(* CODESYS project CtaAppStellAntrieb_1.0.0.3.library
   Description: Stell- Antriebs Library der CTA
   Version: 1.0.0.3
   Title: CtaAppStellAntrieb
   Author: SIS
   Company: CTA
   DocFormat: reStructuredText
   Placeholder: CtaAppStellAntrieb
   DefaultNamespace: CtaAppStellAntrieb
   CompiledLibraryCompatibilityVersion: CODESYS V3.5 SP16 Patch 3
   LanguageModelAttribute: qualified-access-only

Project tree, tasks and I/O mapping:
  libraries: Standard, 3.5.18.0 (System); CtaAppBasic, 1.0.0.0 (CTA); CtaAppBmk, 1.0.0.0 (CTA); CtaAppReport, 1.0.0.0 (CTA); CtaSysConfig, 1.0.0.2 (CTA); VisuDialogs, 3.5.16.20 (System); VisuSymbols, 4.5.0.0 (System); CtaSysMotor, 1.0.0.0 (CTA); CtaVisSymbols, 1.0.0.0 (CTA); CtaAppDumper, 1.0.0.0 (CTA); CtaSysIO, 1.0.0.1 (CTA); CtaAppInfluxLog, 1.0.0.1 (CTA); CtaAppModbusSpezifikation, 1.0.0.0 (CTA); CtaVisHelp, 1.0.0.0 (CTA)
  40 Visualizations/
    COLLECTOR/
      visualisation StellAntrieb_Collector
      visualisation StellAntrieb_Collector_TEMP
      Help Funktionen/
        visualisation SelSort
        visualisation SortPfeil
    ICON/
      StellAntrieb_RIGHT/
        Motor_Right/
          Valve_Mix/
            Above/
              visualisation StellAntrieb_MR_Valve_Mix_RA_CheckEnabled
              visualisation StellAntrieb_MR_Valve_Mix_RA_CheckQuerry
              visualisation StellAntrieb_MR_Valve_Mix_Txt_R_Above
            Below/
              visualisation StellAntrieb_MR_Valve_Mix_RB_CheckEnabled
              visualisation StellAntrieb_MR_Valve_Mix_RB_CheckQuerry
              visualisation StellAntrieb_MR_Valve_Mix_Txt_R_Below
          Valve_Flow/
            Above/
              visualisation StellAntrieb_MR_Valve_Flow_RA_CheckEnabled
              visualisation StellAntrieb_MR_Valve_Flow_RA_CheckQuerry
              visualisation StellAntrieb_MR_Valve_Flow_Txt_R_Above
            Below/
              visualisation StellAntrieb_MR_Valve_Flow_RB_CheckEnabled
              visualisation StellAntrieb_MR_Valve_Flow_RB_CheckQuerry
              visualisation StellAntrieb_MR_Valve_Flow_Txt_R_Below
          Valve_AB_Down/
            Above/
              visualisation StellAntrieb_MR_Valve_AB_Down_RA_CheckQuerry
              visualisation StellAntrieb_MR_Valve_AB_Down_Txt_R_Above
              visualisation StellAntrieb_MR_Valve_AB_Down_RA_CheckEnabled
            Below/
              visualisation StellAntrieb_MR_Valve_AB_Down_Txt_R_Below
              visualisation StellAntrieb_MR_Valve_AB_Down_RB_CheckEnabled
              visualisation StellAntrieb_MR_Valve_AB_Down_RB_CheckQuerry
          Valve_AB_Up/
            Above/
              visualisation StellAntrieb_MR_Valve_AB_Up_RA_CheckEnabled
              visualisation StellAntrieb_MR_Valve_AB_Up_RA_CheckQuerry
              visualisation StellAntrieb_MR_Valve_AB_Up_Txt_R_Above
            Below/
              visualisation StellAntrieb_MR_Valve_AB_Up_RB_CheckEnabled
              visualisation StellAntrieb_MR_Valve_AB_Up_RB_CheckQuerry
              visualisation StellAntrieb_MR_Valve_AB_Up_Txt_R_Below
        Motor_Above/
          Valve_AB_Left/
            visualisation StellAntrieb_MA_Valve_AB_Left_RA_CheckEnabled
            visualisation StellAntrieb_MA_Valve_AB_Left_RA_CheckQuerry
            visualisation StellAntrieb_MA_Valve_AB_Left_Txt_R_Above
          Valve_AB_Right/
            visualisation StellAntrieb_MA_Valve_AB_Right_RA_CheckEnabled
            visualisation StellAntrieb_MA_Valve_AB_Right_RA_CheckQuerry
            visualisation StellAntrieb_MA_Valve_AB_Right_Txt_R_Above
          Valve_Flow/
            visualisation StellAntrieb_MA_Valve_Flow_RA_CheckEnabled
            visualisation StellAntrieb_MA_Valve_Flow_RA_CheckQuerry
            visualisation StellAntrieb_MA_Valve_Flow_Txt_R_Above
          Valve_Mix/
            visualisation StellAntrieb_MA_Valve_Mix_RA_CheckEnabled
            visualisation StellAntrieb_MA_Valve_Mix_RA_CheckQuerry
            visualisation StellAntrieb_MA_Valve_Mix_Txt_R_Above
        Motor_Below/
          Valve_AB_Right/
            visualisation StellAntrieb_MB_Valve_AB_Right_RB_CheckEnabled
            visualisation StellAntrieb_MB_Valve_AB_Right_RB_CheckQuerry
            visualisation StellAntrieb_MB_Valve_AB_Right_Txt_R_Below
          Valve_AB_Left/
            visualisation StellAntrieb_MB_Valve_AB_Left_RB_CheckEnabled
            visualisation StellAntrieb_MB_Valve_AB_Left_RB_CheckQuerry
            visualisation StellAntrieb_MB_Valve_AB_Left_Txt_R_Below
          Valve_Flow/
            visualisation StellAntrieb_MB_Valve_Flow_RB_CheckEnabled
            visualisation StellAntrieb_MB_Valve_Flow_RB_CheckQuerry
            visualisation StellAntrieb_MB_Valve_Flow_Txt_R_Below
          Valve_Mix/
            visualisation StellAntrieb_MB_Valve_Mix_RB_CheckEnabled
            visualisation StellAntrieb_MB_Valve_Mix_RB_CheckQuerry
            visualisation StellAntrieb_MB_Valve_Mix_Txt_R_Below
      StellAntrieb_BASE/
        Ventile/
          DurchflussVentil/
            Motor_Below/
              visualisation MB_Durchgang
            Motor_Above/
              visualisation MA_Durchgang
            Motor_Right/
              visualisation MR_Durchgang
            Motor_Left/
              visualisation ML_Durchgang
          DreiWegVentil/
            Motor_Below/
              visualisation MB_Ventil_AB_L
              visualisation MB_Ventil_Verteiler
              visualisation MB_Ventil_AB_R
            Motor_Above/
              visualisation MA_Ventil_AB_L
              visualisation MA_Ventil_Verteiler
              visualisation MA_Ventil_AB_R
            Motor_Right/
              visualisation MR_Ventil_AB_Up
              visualisation MR_Ventil_Verteiler
              visualisation MR_Ventil_AB_Down
            Motor_Left/
              visualisation ML_Ventil_AB_Down
              visualisation ML_Ventil_Verteiler
              visualisation ML_Ventil_AB_Up
        Icons/
          visualisation Motor
          Motor_Left/
            visualisation Icon_ML_AB_Down
            visualisation Icon_ML_AB_Up
            visualisation Icon_ML_Verteiler
            visualisation Icon_ML_Durchfluss
          Motor_Right/
            visualisation Icon_MR_AB_Down
            visualisation Icon_MR_AB_Up
            visualisation Icon_MR_Durchfluss
            visualisation Icon_MR_Verteiler
          Motor_Below/
            visualisation Icon_MB_AB_L
            visualisation Icon_MB_AB_R
            visualisation Icon_MB_Verteiler
            visualisation Icon_MB_Durchfluss
          Motor_Above/
            visualisation Icon_MA_AB_L
            visualisation Icon_MA_AB_R
            visualisation Icon_MA_Durchfluss
            visualisation Icon_MA_Verteiler
        Value/
          visualisation ValueUpDwn
          visualisation ValueDwnUp
      StellAntrieb_LEFT/
        Motor_LEFT/
          Valve_AB_Down/
            Above/
              visualisation StellAntrieb_ML_Valve_AB_Down_LA_CheckEnabled
              visualisation StellAntrieb_ML_Valve_AB_Down_LA_CheckQuerry
              visualisation StellAntrieb_ML_Valve_AB_Down_Txt_L_Above
            Below/
              visualisation StellAntrieb_ML_Valve_AB_Down_LB_CheckEnabled
              visualisation StellAntrieb_ML_Valve_AB_Down_LB_CheckQuerry
              visualisation StellAntrieb_ML_Valve_AB_Down_Txt_L_Below
          Valve_Mix/
            Above/
              visualisation StellAntrieb_ML_Valve_Mix_LA_CheckEnabled
              visualisation StellAntrieb_ML_Valve_Mix_LA_CheckQuerry
              visualisation StellAntrieb_ML_Valve_Mix_Txt_L_Above
            Below/
              visualisation StellAntrieb_ML_Valve_Mix_LB_CheckEnabled
              visualisation StellAntrieb_ML_Valve_Mix_LB_CheckQuerry
              visualisation StellAntrieb_ML_Valve_Mix_Txt_L_Below
          Valve_Flow/
            Above/
              visualisation StellAntrieb_ML_Valve_Flow_LA_CheckEnabled
              visualisation StellAntrieb_ML_Valve_Flow_LA_CheckQuerry
              visualisation StellAntrieb_ML_Valve_Flow_Txt_L_Above
            Below/
              visualisation StellAntrieb_ML_Valve_Flow_LB_CheckEnabled
              visualisation StellAntrieb_ML_Valve_Flow_LB_CheckQuerry
              visualisation StellAntrieb_ML_Valve_Flow_Txt_L_Below
          Valve_AB_Up/
            Above/
              visualisation StellAntrieb_ML_Valve_AB_Up_LA_CheckEnabled
              visualisation StellAntrieb_ML_Valve_AB_Up_LA_CheckQuerry
              visualisation StellAntrieb_ML_Valve_AB_Up_Txt_L_Above
            Below/
              visualisation StellAntrieb_ML_Valve_AB_Up_LB_CheckEnabled
              visualisation StellAntrieb_ML_Valve_AB_Up_LB_CheckQuerry
              visualisation StellAntrieb_ML_Valve_AB_Up_Txt_L_Below
        Motor_Above/
          Valve_AB_Left/
            visualisation StellAntrieb_MA_Valve_AB_Left_LA_CheckEnabled
            visualisation StellAntrieb_MA_Valve_AB_Left_LA_CheckQuerry
            visualisation StellAntrieb_MA_Valve_AB_Left_Txt_L_Above
          Valve_AB_Right/
            visualisation StellAntrieb_MA_Valve_AB_Right_LA_CheckEnabled
            visualisation StellAntrieb_MA_Valve_AB_Right_Txt_L_Above
            visualisation StellAntrieb_MA_Valve_AB_Right_LA_CheckQuerry
          Valve_Flow/
            visualisation StellAntrieb_MA_Valve_Flow_Txt_L_Above
            visualisation StellAntrieb_MA_Valve_Flow_LA_CheckQuerry
            visualisation StellAntrieb_MA_Valve_Flow_LA_CheckEnabled
          Valve_Mix/
            visualisation StellAntrieb_MA_Valve_Mix_LA_CheckEnabled
            visualisation StellAntrieb_MA_Valve_Mix_LA_CheckQuerry
            visualisation StellAntrieb_MA_Valve_Mix_Txt_L_Above
        Motor_Below/
          Valve_AB_Left/
            visualisation StellAntrieb_MB_Valve_AB_Left_LB_CheckEnabled
            visualisation StellAntrieb_MB_Valve_AB_Left_LB_CheckQuerry
            visualisation StellAntrieb_MB_Valve_AB_Left_Txt_L_Below
          Valve_AB_Right/
            visualisation StellAntrieb_MB_Valve_AB_Right_LB_CheckEnabled
            visualisation StellAntrieb_MB_Valve_AB_Right_LB_CheckQuerry
            visualisation StellAntrieb_MB_Valve_AB_Right_Txt_L_Below
          Valve_Flow/
            visualisation StellAntrieb_MB_Valve_Flow_LB_CheckEnabled
            visualisation StellAntrieb_MB_Valve_Flow_LB_CheckQuerry
            visualisation StellAntrieb_MB_Valve_Flow_Txt_L_Below
          Valve_Mix/
            visualisation StellAntrieb_MB_Valve_Mix_LB_CheckEnabled
            visualisation StellAntrieb_MB_Valve_Mix_LB_CheckQuerry
            visualisation StellAntrieb_MB_Valve_Mix_Txt_L_Below
    POPUP/
      visualisation StellAntrieb_POPUP
      PARAMETER/
        visualisation StellAntrieb_PARAMETER
        visualisation StellAntrieb_ParameterListe
        StellAntrieb_ParameterBase/
          visualisation StellAntrieb_ParameterBase0
          visualisation StellAntrieb_ParameterBase
          visualisation StellAntrieb_ParameterBase2
          visualisation StellAntrieb_ParameterBase1
        StellAntrieb_Fuse/
          visualisation StellAntrieb_ParameterFuses0
          visualisation StellAntrieb_ParameterFuses
        StellAntrieb_IO/
          visualisation StellAntrieb_ParameterIO0
          visualisation StellAntrieb_ParameterIO1
          visualisation StellAntrieb_ParameterIO
          visualisation StellAntrieb_ParameterIO2
          visualisation StellAntrieb_ParameterIO3
          visualisation StellAntrieb_ParameterIO4
        StellAntrieb_InfluxDb/
          visualisation StellAntrieb_ParameterInfluxDb
          visualisation StellAntrieb_ParameterInfluxDb0
        visualisation StellAntrieb_Icon_StellAntrieb
        visualisation StellAntrieb_POPUP_IO_ITF
      visualisation StellAntrieb_PopUpListe
      MANUAL/
        visualisation StellAntrieb_MANUAL
      OVERVIEW/
        visualisation StellAntrieb_OVERVIEW
      BUS/
        visualisation StellAntrieb_BUS
        visualisation StellAntrieb_BUS_SW0_Detail
        visualisation StellAntrieb_BUS_CW0_Detail
        visualisation StellAntrieb_BUS_CS
        visualisation StellAntrieb_BUS_SW1_Detail
        visualisation StellAntrieb_BUS_SW2_Detail
      REPORTS/
        visualisation StellAntrieb_REPORTS
      IO/
        visualisation StellAntrieb_IO0
        visualisation StellAntrieb_IO
        visualisation StellAntrieb_IO1
  30 Program Organization Units/
    function block fbStellAantrieb [ST]: proHandOn, proAuto, proHandOff, proHandOnY, proHardWareHandModulAktive, actConfig, p_scInfluxDb_fbxEnable, p_scActuatorFuse_fbxEnable, p_scActuatorFuse_fbxInputMb, p_scActuatorFuse_fbxDoesAlarm, p_scBase_fbxEnable, p_scBase_fbxControllMb, p_scBase_fbxInvertiert, p_scBase_fbxRegulatet, p_scBase_fbrYMin, p_scBase_fbrYMax, p_scBase_fbxEnStartPosition, p_scBase_fbrYStartPos, p_scBase_fbtStartPosTime, p_scBase_fbrYStopp, p_scBase_fbtYSettingTime, p_scBase_fbxEnDigitalValve, p_scBase_fbrHysteresisDigital, p_scBase_fbrRefIsOpen, p_scBase_fbrRefIsClosed, p_scBase_fbxEnDigitalMonitoring, p_scBase_fbxEnAnalogMonitoring, p_scFuse_fbxEnable, p_scFuse_fbxInputMb, p_scFuse_fbxDoesAlarm, p_scInStellAtRevisionSwitch_fbxEnable, p_scInStellAtRevisionSwitch_fbxInputMb, p_scInStellAtReady_fbxEnable, p_scInStellAtReady_fbxInputMb, p_scInStellAtHand_fbxEnable, p_scInStellAtHand_fbxInputMb, p_scInStellAtRükClosed_fbxEnable, p_scInStellAtRükClosed_fbxInputMb, p_scInStellAtRükClosed_fbxDoesAlarm, p_scInStellAtRükClosed_fbtDelayStart, p_scInStellAtRükClosed_fbtDelayRun, p_scInStellAtRükClosed_fbiTypeOfAck, p_scInStellAtRükClosed_fbiMaxErrorRetryAllowed, p_scInStellAtRükOpen_fbxEnable, p_scInStellAtRükOpen_fbxInputMb, p_scInStellAtRükOpen_fbxDoesAlarm, p_scInStellAtRükOpen_fbtDelayStart, p_scInStellAtRükOpen_fbtDelayRun, p_scInStellAtRükOpen_fbiTypeOfAck, p_scInStellAtRükOpen_fbiMaxErrorRetryAllowed, p_scInStellAtActualPosition_fbxEnable, p_scInStellAtActualPosition_fbxInputMb, p_scInStellAtActualPosition_fbxDoesAlarm, p_scInStellAtActualPosition_fbrMaxDiff, p_scInStellAtActualPosition_fbtDelayStart, p_scInStellAtActualPosition_fbtDelayRun, p_scInStellAtActualPosition_fbiTypeOfAck, p_scInStellAtActualPosition_fbiMaxErrorRetryAllowed, p_scManual_fbxAlowManualOn, p_scManual_fbuiManualState, p_scManual_fbrManualOnY, proRefToRonYDumper, proConfigError, proValveIcon, actMbControll, actMbState, proModbusTest, proModbusStateWord, proModbusControllWord, proIsError, proIsWarning, proIsRegulatet, proIsEnabled, actState, proIsHandOnOrOff, proIsReady, proIsOnY, proRevisionSwitchOk, proStateSymbol, proAnzError, proAnzInfo, proAnzWarning, proITF_REPORTMANAGER, proIsInverted, proRükIsClosed, proRükIsOpen, proOn, metDI_RükIsOpen, proGetDI_RükIsOpen, proNotShowDI_RükIsOpen, proIsOpen_ITF, metDI_RükIsClosed, proGetDI_RükIsClosed, proNotShowDI_RükIsClosed, proIsClosed_ITF, metDI_RevisionSwitchOk, proNotShowDI_RevisionSwitchOk, proGetDI_RevisionSwitchOK, proRevisionSwitch_ITF, proGetDI_FuseOK, metDI_FuseOK, proNotShowDI_FuseOk, proFuse_ITF, metDI_ActuatorHand, proNotShowDI_ActuatorHand, proGetDI_ActuatorHand, proHandModul_ITF, metDI_IsReady, proNotShowDI_Ready, proGetDI_IsReady, proActuatorReady_ITF, proActuatorFuse_ITF, metDI_ActuatorFuseOk, proNotShowDI_ActuatorFuseOk, proGetDI_ActuatorFuseOk, metAI_ActualPosition, proNotShowAI_ActualPosition, proGetAI_ActualPosition, proActualPosition_ITF, proOnY_ITF, metAO_OnY, metDO_xOnAuf, proOnOpen_ITF, proOnClose_ITF, metDO_xOnZu, proOnY, actPrioOfControll, actResetOnDisable, proOnAuf, proOnZu, FB_INIT, proEn, proEnSymbol, actTrendLog, actReport, proAcknowlege, proAvailable, proLockDown
    function block fbStellAntrieb_Collector [ST]: metRegistry, metSortArray, proMin, proMax, proayStellAntriebTabelle, proMissedBuffer, proBufferError, proayStellAntrieb, metGetStellAntriebITF
    function fcGetBigerStringValue [ST]
    Abstracte Bausteine/
      function block fbAntriebTabellenInfo [ST]: proOnAuf, proStateSymbol, proEnSymbol, proIsOn, proIsOnY, proOn, proOnY, proOnZu, proRükIsClosed, proRükIsOpen
    function fcCheckQuerryReturnIcon [ST]
    Visu/
      function fcValveAnimation [ST]
  00000000-0000-0000-0000-000000000000|D:\CoDeSys\LibrariesV3\trunk\Intern\CAA\CAA Template\3.4.0.0 draft\Placeholder.xml
  00000000-0000-0000-0000-000000000000|D:\CoDeSys\LibrariesV3\trunk\Intern\CAA\CAA Template\3.2.0.3 draft\Prefix.pdf
  00000000-0000-0000-0000-000000000000|D:\CoDeSys\LibrariesV3\trunk\Intern\CAA\CAA Template\3.5.2.0 draft\Placeholder.xml
  20 Structs/
    data type scParameter
    STATE/
      data type scInSAtReady
      data type scInSAtRevisionSwitch
      data type scInSAtActualPosition
      data type scInSAtHand
      data type scInSAtRükOpen
      data type scInSAtRükClosed
    BASE/
      data type scBase
    FUSE/
      data type scFuse
      data type scActuatorFuse
    InfluxDb/
      data type scInfluxDb
    MANUAL/
      data type scManual
    data type enIconName
  50 Images/
  10 Documenation/
    global variables VersionHistory
    global variables readMe
  21 Interface/
    interface ITF_STELLANTRIEB: proAuto, proHandOff, proHandOn, proIsRegulatet, proIsError, proIsWarning, proIsEnabled, proIsHandOnOrOff, proIsReady, proHardWareHandModulAktive, proRevisionSwitchOk, proHandOnY, proEn, proGetDI_RükIsOpen, proNotShowDI_RükIsOpen, proIsOpen_ITF, proGetDI_ActuatorHand, proNotShowDI_ActuatorHand, proHandModul_ITF, proGetDI_ActuatorFuseOk, proNotShowDI_ActuatorFuseOk, proActuatorFuse_ITF, proGetDI_IsReady, proNotShowDI_Ready, proActuatorReady_ITF, proGetDI_FuseOK, proNotShowDI_FuseOk, proFuse_ITF, proGetDI_RevisionSwitchOK, proNotShowDI_RevisionSwitchOk, proRevisionSwitch_ITF, proNotShowAI_ActualPosition, proGetAI_ActualPosition, proActualPosition_ITF, proGetDI_RükIsClosed, proNotShowDI_RükIsClosed, proIsClosed_ITF, proOnOpen_ITF, proOnClose_ITF, proOnY_ITF, proAnzWarning, proITF_REPORTMANAGER, proAnzInfo, proAnzError, proModbusTest, proModbusStateWord, proModbusControllWord, proConfigError, p_scActuatorFuse_fbxEnable, p_scActuatorFuse_fbxInputMb, p_scActuatorFuse_fbxDoesAlarm, p_scBase_fbxEnable, p_scBase_fbxControllMb, p_scBase_fbxInvertiert, p_scBase_fbxRegulatet, p_scBase_fbrYMin, p_scBase_fbrYMax, p_scBase_fbxEnStartPosition, p_scBase_fbrYStartPos, p_scBase_fbtStartPosTime, p_scBase_fbrYStopp, p_scBase_fbtYSettingTime, p_scBase_fbxEnDigitalValve, p_scBase_fbrHysteresisDigital, p_scBase_fbrRefIsOpen, p_scBase_fbrRefIsClosed, p_scBase_fbxEnDigitalMonitoring, p_scBase_fbxEnAnalogMonitoring, p_scFuse_fbxEnable, p_scFuse_fbxInputMb, p_scFuse_fbxDoesAlarm, p_scInStellAtRevisionSwitch_fbxEnable, p_scInStellAtRevisionSwitch_fbxInputMb, p_scInStellAtReady_fbxEnable, p_scInStellAtReady_fbxInputMb, p_scInStellAtHand_fbxEnable, p_scInStellAtHand_fbxInputMb, p_scInStellAtRükClosed_fbxEnable, p_scInStellAtRükClosed_fbxInputMb, p_scInStellAtRükClosed_fbxDoesAlarm, p_scInStellAtRükClosed_fbtDelayStart, p_scInStellAtRükClosed_fbtDelayRun, p_scInStellAtRükClosed_fbiTypeOfAck, p_scInStellAtRükClosed_fbiMaxErrorRetryAllowed, p_scInStellAtRükOpen_fbxEnable, p_scInStellAtRükOpen_fbxInputMb, p_scInStellAtRükOpen_fbxDoesAlarm, p_scInStellAtRükOpen_fbtDelayStart, p_scInStellAtRükOpen_fbtDelayRun, p_scInStellAtRükOpen_fbiTypeOfAck, p_scInStellAtRükOpen_fbiMaxErrorRetryAllowed, p_scInStellAtActualPosition_fbxEnable, p_scInStellAtActualPosition_fbxInputMb, p_scInStellAtActualPosition_fbxDoesAlarm, p_scInStellAtActualPosition_fbrMaxDiff, p_scInStellAtActualPosition_fbtDelayStart, p_scInStellAtActualPosition_fbtDelayRun, p_scInStellAtActualPosition_fbiTypeOfAck, p_scInStellAtActualPosition_fbiMaxErrorRetryAllowed, p_scManual_fbxAlowManualOn, p_scManual_fbuiManualState, p_scManual_fbrManualOnY, p_scInfluxDb_fbxEnable, proRefToRonYDumper, proIsInverted, proValveIcon, proAcknowlege, proAvailable, proLockDown, proOn
    interface ITF_STELLANTRIEB_COLLECTOR: metSortArray, proayStellAntriebTabelle, proMax, proMin, proBufferError, proMissedBuffer, metGetStellAntriebITF
    interface ITF_STELLANTRIEB_TABELLE_INFO: proRükIsOpen, proRükIsClosed, proStateSymbol, proEnSymbol, proOnZu, proIsOnY, proOnAuf, proOnY
  11 Library Parameter/
    global variables Parameter
  12 Konstanten/
    global variables GlobalKonstant
  60 Textlisten/
    text list Error
    text list Info
    text list Warnung
  13 Globale Variablen/
    global variables GVL_StellAntrieb
  text list GlobalTextList
  5ce3da45-db07-42e7-a21c-a00fff4ed8f6|C:\Users\sis\Downloads\dip-switch.svg
  5ce3da45-db07-42e7-a21c-a00fff4ed8f6|C:\Users\sis\Downloads\lightning-bolt-circle.svg
  5ce3da45-db07-42e7-a21c-a00fff4ed8f6|C:\Users\sis\Downloads\sine-wave.svg
  5ce3da45-db07-42e7-a21c-a00fff4ed8f6|C:\Users\sis\Downloads\eye.svg
  5ce3da45-db07-42e7-a21c-a00fff4ed8f6|C:\Users\sis\Downloads\lan.svg
*)

// 20 Structs/scParameter
{attribute 'pack_mode' := '1'} 
TYPE scParameter :
    STRUCT
        scBase              	:   scBase;
        scFuse              	:   scFuse;
        scActuatorFuse         	:   scActuatorFuse;
        scInSAtRevisionSwitch	:   scInSAtRevisionSwitch;
        scInSAtReady         	:   scInSAtReady; 
        scInSAtActualPosition   :   scInSAtActualPosition;
		scInSAtRükOpen			:	scInSAtRükOpen;
		scInSAtRükClosed		:	scInSAtRükClosed;
        scManual            	:   scManual;
        scInfluxDb          	:   scInfluxDb;
        scInSAtHand          	:   scInSAtHand;
    END_STRUCT
END_TYPE

// 20 Structs/STATE/scInSAtReady
{attribute 'pack_mode' := '1'} 
TYPE scInSAtReady :
    STRUCT
        fbxEnable                    : CtaSysConfig.fbBOOL;
        fbxInputMb                   : CtaSysConfig.fbBOOL;          
    END_STRUCT
END_TYPE

// 20 Structs/STATE/scInSAtRevisionSwitch
{attribute 'pack_mode' := '1'} 
TYPE scInSAtRevisionSwitch :
    STRUCT
        fbxEnable                   : CtaSysConfig.fbBOOL;
        fbxInputMb                  : CtaSysConfig.fbBOOL;           
    END_STRUCT
END_TYPE

// 20 Structs/STATE/scInSAtActualPosition
{attribute 'pack_mode' := '1'} 
TYPE scInSAtActualPosition :
    STRUCT
        fbxEnable                    : CtaSysConfig.fbBOOL;
        fbxInputMb                   : CtaSysConfig.fbBOOL;   
        fbxDoesAlarm                 : CtaSysConfig.fbBOOL;  
        fbrMaxDiff                   : CtaSysConfig.fbREAL;
        fbtDelayStart                : CtaSysConfig.fbTIME;
        fbtDelayRun                  : CtaSysConfig.fbTIME;
		fbiTypeOfAck               	 : CtaSysConfig.fbINT;   
        fbiMaxErrorRetryAllowed      : CtaSysConfig.fbINT;         
    END_STRUCT
END_TYPE

// 20 Structs/STATE/scInSAtHand
{attribute 'pack_mode' := '1'} 
TYPE scInSAtHand :
    STRUCT
        fbxEnable                   : CtaSysConfig.fbBOOL;    
        fbxInputMb                  : CtaSysConfig.fbBOOL; 
    END_STRUCT
END_TYPE

// 20 Structs/BASE/scBase
{attribute 'pack_mode' := '1'} 
TYPE scBase :
    STRUCT
        fbxEnable       		:   CtaSysConfig.fbBOOL;
		fbxRegulatet    		:   CtaSysConfig.fbBOOL;
		fbxControllMb   		:   CtaSysConfig.fbBOOL;
		fbxInvertiert			:	CtaSysConfig.fbBOOL;
		fbrYMin         		:   CtaSysConfig.fbREAL;
        fbrYMax         		:   CtaSysConfig.fbREAL;
		fbxEnStartPosition		:	CtaSysConfig.fbBOOL;
		fbrYStartPos			:	CtaSysConfig.fbREAL;
		fbtStartPosTime			:	CtaSysConfig.fbTIME;
		fbrYStopp				:	CtaSysConfig.fbREAL;		
		fbtYSettingTime			:	CtaSysConfig.fbTIME;
		fbxEnDigitalValve		:	CtaSysConfig.fbBOOL;		
		fbrHysteresisDigital	:	CtaSysConfig.fbREAL;		
		fbrRefIsOpen			:	CtaSysConfig.fbREAL;
		fbrRefIsClosed			:	CtaSysConfig.fbREAL;
		fbxEnDigitalMonitoring	:	CtaSysConfig.fbBOOL;
		fbxEnAnalogMonitoring	:	CtaSysConfig.fbBOOL;		
    END_STRUCT
END_TYPE

// 20 Structs/FUSE/scFuse
{attribute 'pack_mode' := '1'} 
TYPE scFuse :
    STRUCT
        fbxEnable               : CtaSysConfig.fbBOOL;
        fbxInputMb              : CtaSysConfig.fbBOOL;
        fbxDoesAlarm            : CtaSysConfig.fbBOOL;
    END_STRUCT
END_TYPE

// 20 Structs/FUSE/scActuatorFuse
{attribute 'pack_mode' := '1'} 
TYPE scActuatorFuse :
    STRUCT
        fbxEnable             : CtaSysConfig.fbBOOL;
        fbxInputMb            : CtaSysConfig.fbBOOL;
        fbxDoesAlarm          : CtaSysConfig.fbBOOL;      
    END_STRUCT
END_TYPE

// 20 Structs/InfluxDb/scInfluxDb
{attribute 'pack_mode' := '1'} 
TYPE scInfluxDb :
    STRUCT
        fbxEnable       :   CtaSysConfig.fbBOOL;
    END_STRUCT
END_TYPE

// 20 Structs/MANUAL/scManual
{attribute 'pack_mode' := '1'} 
TYPE scManual :
    STRUCT
        fbxAlowManualOn         : CtaSysConfig.fbBOOL;    
        fbuiManualState         : CtaSysConfig.fbUINT;            // 0 = Auto ; 1 = Manual Off 2 = Manual On
        fbrManualOnY            : CtaSysConfig.fbREAL; 
    END_STRUCT
END_TYPE

// 20 Structs/STATE/scInSAtRükOpen
TYPE scInSAtRükOpen :
	STRUCT
		fbxEnable                    : CtaSysConfig.fbBOOL;
		fbxInputMb                   : CtaSysConfig.fbBOOL;   
		fbxDoesAlarm                 : CtaSysConfig.fbBOOL;  
		fbtDelayStart                : CtaSysConfig.fbTIME;
		fbtDelayRun                  : CtaSysConfig.fbTIME;
		fbiTypeOfAck               	 : CtaSysConfig.fbINT;   
        fbiMaxErrorRetryAllowed      : CtaSysConfig.fbINT;      
	END_STRUCT
END_TYPE

// 20 Structs/STATE/scInSAtRükClosed
TYPE scInSAtRükClosed :
	STRUCT
		fbxEnable                    : CtaSysConfig.fbBOOL;
		fbxInputMb                   : CtaSysConfig.fbBOOL;   
		fbxDoesAlarm                 : CtaSysConfig.fbBOOL;  
		fbtDelayStart                : CtaSysConfig.fbTIME;
		fbtDelayRun                  : CtaSysConfig.fbTIME;
		fbiTypeOfAck                 : CtaSysConfig.fbINT;   
        fbiMaxErrorRetryAllowed      : CtaSysConfig.fbINT;    
	END_STRUCT
END_TYPE

// 20 Structs/enIconName
{attribute 'qualified_only'}
{attribute 'strict'}
TYPE enIconName :
(
	S_AT_MA_Valve_AB_Left_Txt_L_Above := 1,
	S_AT_MA_Valve_AB_Right_Txt_L_Above,
	S_AT_MA_Valve_Flow_Txt_L_Above,
	S_AT_MA_Valve_Mix_Txt_L_Above,
	S_AT_MB_Valve_AB_Left_Txt_L_Below,
	S_AT_MB_Valve_AB_Right_Txt_L_Below,
	S_AT_MB_Valve_Flow_Txt_L_Below,
	S_AT_MB_Valve_Mix_Txt_L_Below,
	S_AT_ML_Valve_AB_Down_Txt_L_Above,
	S_AT_ML_Valve_AB_Down_Txt_L_Below,
	S_AT_ML_Valve_AB_Up_Txt_L_Above,
	S_AT_ML_Valve_AB_Up_Txt_L_Below,
	S_AT_ML_Valve_Flow_Txt_L_Above,
	S_AT_ML_Valve_Flow_Txt_L_Below,
	S_AT_ML_Valve_Mix_Txt_L_Above,
	S_AT_ML_Valve_Mix_Txt_L_Below,
	S_AT_MA_Valve_AB_Left_Txt_R_Above,
	S_AT_MA_Valve_AB_Right_Txt_R_Above,
	S_AT_MA_Flap_Txt_R_Above,
	S_AT_MA_Valve_Flow_Txt_R_Above,
	S_AT_MA_Valve_Mix_Txt_R_Above,
	S_AT_MB_Valve_AB_Left_Txt_R_Below,
	S_AT_MB_Valve_AB_Right_Txt_R_Below,
	S_AT_MB_Valve_Flow_Txt_R_Below,
	S_AT_MB_Valve_Mix_Txt_R_Below,
	S_AT_MR_Valve_AB_Down_Txt_R_Above,
	S_AT_MR_Valve_AB_Down_Txt_R_Below,
	S_AT_MR_Valve_AB_Up_Txt_R_Above,
	S_AT_MR_Valve_AB_Up_Txt_R_Below,
	S_AT_MR_Valve_Flow_Txt_R_Above,
	S_AT_MR_Valve_Flow_Txt_R_Below,
	S_AT_MR_Valve_Mix_Txt_R_Above,
	S_AT_MR_Valve_Mix_Txt_R_Below
	
);
END_TYPE

// 10 Documenation/VersionHistory
(* 

.. image:: ../../Images/CTA_Logo.jpg
   :align: right
   :width: 15% 

**Vorlage**   


============ =========== =========== ============================================
**Date**     **Version** **Author**  **Change**
------------ ----------- ----------- --------------------------------------------
04.03.2021   0.0.0.0     SIS         Vorlage erstellt

============ =========== =========== ============================================


*)
VAR_GLOBAL
    stInfo : STRING:= '0.0.0.0, Vorlage, CTA';
END_VAR

// 10 Documenation/readMe
(*

**ReadMe**
 
|	**Empfehlung**
|
|	Biblitothek CtaAppStellAntrieb zur Ansteuerung von Stellantrieben
|	Instanzieren Sie den CtaAppStellAntrieb.fbStellAntrieb in ihrem Funktionsbaustein oder POU beispielsweise als fbStelAX. (X = Nr.) 
|	Deklarieren Sie die Struktur Variable welche als Parameter und zur ansteuerung dienen wie im Code beispiel.
|  
| *Beispiel* 

+-----------------------+---------------------------------------------------------------------------------------------------------------------------------------------------------------------------------------------------------------------------------------------------------------------------------------------------------------------------------------------------------------------------------------------------------------------------------------+
| Beschreibung          |  Code                                                                                                                                                                                                                                                                                                                                                                                                                                 |
+=======================+=======================================================================================================================================================================================================================================================================================================================================================================================================================================+
| Pou oder SmFb         | .. code-block:: codesys                                                                                                                                                                                                                                                                                                                                                                                                               |
|                       |                                                                                                                                                                                                                                                                                                                                                                                                                                       |
|                       |	// Deklaration als VAR im POU oder dem selbsterstellten Funktionsbaustein                                                                                                                                                                                                                                                                                                                                                        	|
|                       |   VAR   																																																				 																																																				|
|						|	    (*Stellantrieb 1*)																																																		 																																																		|
|						|		fbStelA1			: CtaAppStellAntrieb.fbStellAntrieb;                                                                                                                                                                                                                                                                                                                                                               			|
|                       | 		(*Stellantrieb 2*)																																																		 																																																		|
|			 			|		fbStelA2			: CtaAppStellAntrieb.fbStellAntrieb;																																												 																																														|
|			 			|	END_VAR                                                                                                                                                                                                                                                                                                                                                                                                                          	|
+-----------------------+---------------------------------------------------------------------------------------------------------------------------------------------------------------------------------------------------------------------------------------------------------------------------------------------------------------------------------------------------------------------------------------------------------------------------------------+
| Code für Init         | .. code-block:: codesys                                                                                                                                                                                                                                                                                                                                                                                                               |
|                       |   																																																					 																																																				|
|			 			|	// Kopieren des nachfolgenden Codes in eine Action zur Initialisierung der Parameter. Zum Beispiel actConfig.																																																				 																										|
|                       |	{region "Parameter Stellantrieb 1"}                                                                                                                                                                                                                                                                                                                                                                                                 |
|			 			|		(*Basis*)                                                                                                                                                                                                                                                                                                                                                                                                                       |
|						|		fbStelA1.scParameter.scBase.fbxEnable                				(_WertInit :=  TRUE																		 );		//P1 Ein- Ausschalten des Stellantriebs                                                                                                                                                                                                           			|
|						|		fbStelA1.scParameter.scBase.fbxRegulatet 							(_WertInit :=  TRUE																		 );     //P2 Stellantrieb ist geregelt / nicht geregelt                                                                                                                                                                                            					|
|						|		fbStelA1.scParameter.scBase.fbxControllMb 							(_WertInit := FALSE																		 );     //P3 Ansteuerung oder Signalauswertung über Modbus                                                                                                                                                                                            				|
|						|		fbStelA1.scParameter.scBase.fbxInvertiert							(_WertInit := FALSE																		 );     //P4 Stellantrieb Invertierung                                                                                                                                                                                                                  			|
|						|		fbStelA1.scParameter.scBase.fbrYMin    								(_WertInit :=   0.0									, _minInit :=      , _maxInit:=      );     //P5 Minimal zulässiger Stellwert des Stellantriebs                                                                                                                                                   	 													|
|						|		fbStelA1.scParameter.scBase.fbrYMax    								(_WertInit :=   0.0									, _minInit :=      , _maxInit:=      );     //P6 Maximal zulässiger Stellwert des Stellantriebs																																																			|
|						|		fbStelA1.scParameter.scBase.fbxEnStartPosition 						(_WertInit :=  TRUE																		 );     //P7 Wenn aktiviert fährt Stellantreieb bei anstehender Fraigabe an definierte Position                                                                                                                                                                     |
|						|		fbStelA1.scParameter.scBase.fbrYStartPos    						(_WertInit :=   0.0									, _minInit :=      , _maxInit:=      );     //P8 Parameter zur Einstellung der Startposition                                                                                                                                                  	 														|
|						|		fbStelA1.scParameter.scBase.fbtStartPosTime							(_WertInit :=  T#0S									, _minInit :=      , _maxInit:= 	 );     //P9 Zeit zur Einstellung wie lange Stellantrieb an der Startposition verharren soll                                                                                                                                                                        |
|						|		fbStelA1.scParameter.scBase.fbrYStopp    							(_WertInit :=   0.0									, _minInit :=      , _maxInit:=      );     //P10 Parameter zur Einstellung der Stopposition                                                                                                                                                   	 														|
|						|		fbStelA1.scParameter.scBase.fbtYSettingTime							(_WertInit :=  T#0S									, _minInit :=      , _maxInit:= 	 );     //P11 Stellzeit des Stellantriebs                                                                                                                                                                                                                           |
|						|		fbStelA1.scParameter.scBase.fbxEnDigitalValve 						(_WertInit := FALSE																		 );     //P12 Aktivierung, Deaktivierung der digitalen Ansteuerung                                                                                                                                                                                            		|
|						|		fbStelA1.scParameter.scBase.fbrHysteresisDigital    				(_WertInit :=   0.0									, _minInit :=      , _maxInit:=      );     //P13 Einstellbare Hysterese für die digitale Ansteuerung                                                                                                                                                  	 												|
|						|		fbStelA1.scParameter.scBase.fbrRefIsOpen    						(_WertInit :=   0.0									, _minInit :=      , _maxInit:=      );     //P14 Parameter zur einstellung des Referenzwertes bei welchem von einem offenen Stellantrieb ausgegangen wird                                                                                                                                              |
|						|		fbStelA1.scParameter.scBase.fbrRefIsClosed    						(_WertInit :=   0.0									, _minInit :=      , _maxInit:=      );     //P15 Parameter zur einstellung des Referenzwertes bei welchem von einem geschlossenen Stellantrieb ausgegangen wird                                                                                                                                        |
|						|		fbStelA1.scParameter.scBase.fbxEnDigitalMonitoring 					(_WertInit := FALSE																		 );     //P16 Aktivierung der digitalen Überwachung                                                                                                                                                                                            						|
|						|		fbStelA1.scParameter.scBase.fbxEnAnalogMonitoring					(_WertInit := FALSE																		 );     //P17 Aktivierung der analogen Überwachung                                                                                                                                                                                                                  |
|						|		(* Fuse Parameter *)                                                                                                                                                                                                                                                                                                                                                                                          					|
|						|		fbStelA1.scParameter.scFuse.fbxEnable   							(_WertInit := FALSE																		 );     //P18 Sicherung ist vorhanden / nicht vorhanden                                                                                                                                          																	|
|						|		fbStelA1.scParameter.scFuse.fbxInputMb  							(_WertInit := FALSE																		 );     //P19 Ansteuerung oder Signalauswertung über Modbus                                                                                                                                                                                                      	|
|						|		fbStelA1.scParameter.scFuse.fbxDoesAlarm							(_WertInit := FALSE																		 );     //P20 Abfallendes Signal löst Fehler aus                                                                                                                                                                                                   					|
|						|		(* Stellantrieb Fuse Parameter *)       																																																																																														|
|						|		fbStelA1.scParameter.scActuatorFuse.fbxEnable                   	(_WertInit := FALSE																		 );     //P21 Leistungsschutzschalter ist vorhanden / nicht vorhanden                                                                                                                                                                                            	|
|						|		fbStelA1.scParameter.scActuatorFuse.fbxInputMb   					(_WertInit := FALSE																		 );     //P22 Ansteuerung oder Signalauswertung über Modbus                                                                                                                                                                                                      	|
|						|		fbStelA1.scParameter.scActuatorFuse.fbxDoesAlarm 					(_WertInit := FALSE																		 );     //P23 Abfallendes Signal löst Fehler aus                                                                                                                                                                                                                	|
|						|		(* Revision Switch Parameter *)                                 		                                                                                                                                                                                                                                                                                                                                                        |
|						|		fbStelA1.scParameter.scInSAtRevisionSwitch.fbxEnable  				(_WertInit := FALSE																		 );     //P24 Revisionschalter ist vorhanden / nicht vorhanden                                                                                                                                                                         								|
|						|		fbStelA1.scParameter.scInSAtRevisionSwitch.fbxInputMb 				(_WertInit := FALSE																		 );     //P25 Ansteuerung oder Signalauswertung über Modbus                                                                                                                                                                                                     	|
|						|		(* Ready Input Parameter *)                                                                                                                                                                                                                                                                                                                                                                                                     |
|						|		fbStelA1.scParameter.scInSAtReady.fbxEnable  						(_WertInit := FALSE																		 );     //P26 Readysignal ist vorhanden / nicht vorhanden                                                                                                                                                                                                       	|
|						|		fbStelA1.scParameter.scInSAtReady.fbxInputMb 						(_WertInit := FALSE																		 );     //P27 Ansteuerung oder Signalauswertung über Modbus                                                                                                                                                                                                     	|
|						|		(* Stellantrieb Input Hand *)         							                                                                                                                                                                                                                                                                                                                                                                |
|						|		fbStelA1.scParameter.scInSAtHand.fbxEnable 							(_WertInit := FALSE																		 );     //P28 Handmodul ist vorhanden / nicht vorhanden                                                                                                                                                                                                        		|
|						|		fbStelA1.scParameter.scInSAtHand.fbxInputMb							(_WertInit := FALSE																		 );     //P29 Ansteuerung oder Signalauswertung über Modbus                                                                                                                                                                                                    		|
|						|		(* Is closed Input Parameter *)                     	        	                                                                                                                                                                                                                                                                                                                                                            |
|						|		fbStelA1.scParameter.scInSAtRükClosed.fbxEnable		 				(_WertInit := FALSE																		 );     //P30 Rückmeldung ZU ist vorhanden / nicht vorhanden                                                                                                                                                                                                    	|
|						|		fbStelA1.scParameter.scInSAtRükClosed.fbxInputMb      				(_WertInit := FALSE																		 );     //P31 Ansteuerung oder Signalauswertung über Modbus                                                                                                                                                                                                     	|
|						|		fbStelA1.scParameter.scInSAtRükClosed.fbxDoesAlarm    				(_WertInit := FALSE																		 );     //P32 Fehlendes oder abfallendes Signal löst Fehler aus                                                                                                                                                             										|
|						|		fbStelA1.scParameter.scInSAtRükClosed.fbtDelayStart   				(_WertInit :=  T#0S									, _minInit :=      , _maxInit:= 	 );     //P33 Verzögerung der Fehlerausgabe nach Start                                                                                                                                                                                                          	|
|						|		fbStelA1.scParameter.scInSAtRükClosed.fbtDelayRun     				(_WertInit :=  T#0S									, _minInit :=      , _maxInit:= 	 );     //P34 Verzögerung der Fehlerausgabe während Betrieb                                                                                                                                                                                                     	|
|						|		fbStelA1.scParameter.scInSAtRükClosed.fbiTypeOfAck					(_WertInit :=     0									, _minInit :=     0, _maxInit:=     2);     //P35 Art der Quittierung des Fehlers (auto, quittierned, quittiernd bis n meldung)                                                                                                                                                                     	|
|						|		fbStelA1.scParameter.scInSAtRükClosed.fbiMaxErrorRetryAllowed		(_WertInit :=     3									, _minInit :=     0, _maxInit:= 	5);     //P36 Maximale Anzahl Wiederholungen bis zu Sperrung der Anlage                                                                                                                                                                           					|
|						|		(* Is open Input Parameter *)                       			                                                                                                                                                                                                                                                                                                                                                                |
|						|		fbStelA1.scParameter.scInSAtRükOpen.fbxEnable		 				(_WertInit := FALSE																		 );     //P37 Rückmeldung OFFEN ist vorhanden / nicht vorhanden                                                                                                                                                                                                 	|
|						|		fbStelA1.scParameter.scInSAtRükOpen.fbxInputMb        				(_WertInit := FALSE																		 );     //P38 Ansteuerung oder Signalauswertung über Modbus                                                                                                                                                                                                    		|
|						|		fbStelA1.scParameter.scInSAtRükOpen.fbxDoesAlarm      		    	(_WertInit := FALSE																		 );     //P39 Fehlendes oder abfallendes Signal löst Fehler aus                                                                                                                                                                                                		|
|						|		fbStelA1.scParameter.scInSAtRükOpen.fbtDelayStart     				(_WertInit :=  T#0S									, _minInit :=      , _maxInit:= 	 );     //P40 Verzögerung der Fehlerausgabe nach Start                                                                                                                                                                                                         		|
|						|		fbStelA1.scParameter.scInSAtRükOpen.fbtDelayRun       				(_WertInit :=  T#0S									, _minInit :=      , _maxInit:= 	 );     //P41 Verzögerung der Fehlerausgabe während Betrieb                                                                                                                                                                                                    		|
|						|		fbStelA1.scParameter.scInSAtRükOpen.fbiTypeOfAck					(_WertInit :=     0									, _minInit :=     0, _maxInit:=     2);     //P42 Art der Quittierung des Fehlers  (auto, quittierned, quittiernd bis n meldung)                                                                                                                                                                    	|
|						|		fbStelA1.scParameter.scInSAtRükOpen.fbiMaxErrorRetryAllowed			(_WertInit :=     3									, _minInit :=     0, _maxInit:= 	5);     //P43 Maximale Anzahl Wiederholungen bis zu Sperrung der Anlage                                                                                                                                                                                      		|
|						|		(* Actual value Input Parameter *)                          	                                                                                                                                                                                                                                                                                                                                                                |
|						|		fbStelA1.scParameter.scInSAtActualPosition.fbxEnable     			(_WertInit := FALSE																		 );     //P44 Rückmeldung des Istwerts ist vorhanden / nicht vorhanden                                                                                                                                                                                          	|
|						|		fbStelA1.scParameter.scInSAtActualPosition.fbxInputMb    			(_WertInit := FALSE																		 );     //P45 Ansteuerung oder Signalauswertung über Modbus                                                                                                                                                                                                   		|
|						|		fbStelA1.scParameter.scInSAtActualPosition.fbxDoesAlarm  			(_WertInit := FALSE																		 );     //P46 Unter oder überschreitung der Maximal erlaubten Differenz löst Fehler aus                                                                                                                                                            					|
|						|		fbStelA1.scParameter.scInSAtActualPosition.fbrMaxDiff    			(_WertInit :=   0.0									, _minInit :=      , _maxInit:=      );     //P47 Maximal erlaubte Differenz des Stell- zum Istwert                                                                                                                                                   	 												|
|						|		fbStelA1.scParameter.scInSAtActualPosition.fbtDelayStart 			(_WertInit :=  T#0S									, _minInit :=      , _maxInit:= 	 );     //P48 Verzögerung der Fehlerausgabe nach Start                                                                                                                                        					  													|
|						|		fbStelA1.scParameter.scInSAtActualPosition.fbtDelayRun   			(_WertInit :=  T#0S									, _minInit :=      , _maxInit:= 	 );     //P49 Verzögerung der Fehlerausgabe während Betrieb                                                                                                                                               															|
|						|		fbStelA1.scParameter.scInSAtActualPosition.fbiTypeOfAck				(_WertInit :=     0									, _minInit :=     0, _maxInit:=     2);     //P50 Art der Quittierung des Fehlers (auto, quittierned, quittiernd bis n meldung)                                                                                                       																	|
|						|		fbStelA1.scParameter.scInSAtActualPosition.fbiMaxErrorRetryAllowed	(_WertInit :=     3									, _minInit :=     0, _maxInit:= 	5);     //P51 Maximale Anzahl Wiederholungen bis zu Sperrung der Anlage                                                                                                                                   															|
|						|		(*Sollwertdämpfung*)																																																																																																			|
|						|		fbStelA1.fbDumperRonY.scParameter.fbrTup							(_wertInit :=   1.0                                 , _minInit :=       , _maxInit :=    );      //P34 Maximal erlaubte Differenz des Stell- zum Istwert																																																	|
|						|		fbStelA1.fbDumperRonY.scParameter.fbrTdown							(_wertInit :=   1.0                                 , _minInit :=       , _maxInit :=    );      //P34 Maximal erlaubte Differenz des Stell- zum Istwert																																																	|
|						|		fbStelA1.fbDumperRonY.scParameter.fbrBand							(_wertInit := 100.0                                 , _minInit :=       , _maxInit :=    );      //P34 Maximal erlaubte Differenz des Stell- zum Istwert																																																	|
|						|		fbStelA1.fbDumperRonY.scParameter.fbxInExpOut						(_wertInit := FALSE                                                                      );      //P42 Handansteuerung zulassen / nicht zulassen																																																			|
|						|		(* InfluxDb *)                                                                                                                                                                                                                                                                                                                                                                                                                  |
|						|		fbStelA1.scParameter.scInfluxDb.fbxEnable                           (_WertInit := FALSE																		 );     //P52 Aktivierung / Deaktivierung der Trenddaten                                                                                                                                                                                                     		|
|						|		(* Manual Parameter *)                                                                                                                                                                                                                                                                                                                                                                                                          |
|						|		fbStelA1.scParameter.scManual.fbxAlowManualOn                       (_WertInit := FALSE																		 );     //P53 Handansteuerung zulassen / nicht zulassen                                                                                                                                                                                                       		|
|						|		fbStelA1.scParameter.scManual.fbuiManualState                       (_WertInit :=     0									, _minInit :=     0, _maxInit:=     2);     //P54 Ansteuerungsmodus der Klappe (auto, manuell, gesperrt)                                                                                                                                                                             					|
|						|		fbStelA1.scParameter.scManual.fbrManualOnY	                      	(_WertInit :=     0									, _minInit :=      , _maxInit:=      );     //P55 Stellwert für Stellantrieb                                                                                                                                                                                             								|
|						|	{endregion} 	                                                                                                                                                                                                                                                                     																																				|
+-----------------------+---------------------------------------------------------------------------------------------------------------------------------------------------------------------------------------------------------------------------------------------------------------------------------------------------------------------------------------------------------------------------------------------------------------------------------------+
*)                                                                                                                                                                                                                                                                                                                                                                                                                                                               
VAR_GLOBAL
	xReadMeDone              :   BOOL; 
END_VAR

// 13 Globale Variablen/GVL_StellAntrieb
{attribute 'qualified_only'}
VAR_GLOBAL
    fbStellAntrieb_Collector  :   fbStellAntrieb_Collector;   
    xValidData      :   BOOL;
END_VAR

// 11 Library Parameter/Parameter
{attribute 'qualified_only'}
VAR_GLOBAL CONSTANT
    iMaxStellAntrieb :   INT   := 60;         // Maximale Anzahl verwendeter AT-Bausteine    
END_VAR

// 12 Konstanten/GlobalKonstant
{attribute 'qualified_only'}
VAR_GLOBAL CONSTANT 	
	stReportTextListError   : CtaAppReport.stReportTextList := 'CtaAppStellAntrieb.Error';
	stReportTextListWarning : CtaAppReport.stReportTextList := 'CtaAppStellAntrieb.Warnung';
	stReportTextListInfo    : CtaAppReport.stReportTextList := 'CtaAppStellAntrieb.Info';	
    uiMaxParameter          : UINT := 55;
END_VAR

// 30 Program Organization Units/fbStellAantrieb
FUNCTION_BLOCK fbStellAantrieb EXTENDS fbAntriebTabellenInfo IMPLEMENTS ITF_STELLANTRIEB 
VAR_INPUT
    xRelease                    	:   BOOL;
    rRelease                    	:   REAL;	
END_VAR                         
VAR_OUTPUT                      
    (* Commmands *)	
	xOnAuf							:	BOOL;	
	xOnZu							:	BOOL;	
    rOnY                        	:   REAL; 	// Stellantrieb Position
	
	(* Status Outputs*)
	xIsOpen							:	BOOL;
	xIsClose						:	BOOL;
END_VAR                 
VAR 
	uiValveIcon						:	UINT;                    
    (* State Intern *)      	
    scEWI                       	:   CtaAppReport.scReportNr;
	xOn								:	BOOL;                
    xIsWarning                  	:   BOOL;
    _xIsWarning                 	:   BOOL;	
    xIsError                    	:   BOOL;
    _xIsError                   	:   BOOL;	
    xIsRegulatet                	:   BOOL;	
    xIsEnabled                  	:   BOOL;
    xIsHand                     	:   BOOL;
    xIsHandOn                   	:   BOOL;
    xIsHandOff                  	:   BOOL;
    xIsAuto                     	:   BOOL;
	xIsInverted						:	BOOL;   
    xConfigError                	:   BOOL;
	fbDumperRonY				:	CtaAppDumper.fbDumper;
	(* ITF OUT*)
	ITF_xOnAuf						:	CtaSysIO.ITF_IO;	
	ITF_xOnZu						:	CtaSysIO.ITF_IO;
	ITF_rOnY						:	CtaSysIO.ITF_IO;	
    (* Inputs *)
	(* Aktuelle Position *)
	rActualPosition					:	REAL;	
	rInActualPosition				:	REAL;
	rInActualPositionMb				:	REAL;
	ITF_ActualPosition				:	CtaSysIO.ITF_IO;
	(* Rückmeldung offen *)
	xRückIsOpen						:	BOOL;	
	xInRükIsOpen					:	BOOL;
	xInRükIsOpenMb					:	BOOL;
	ITF_RükIsOpen					:	CtaSysIO.ITF_IO;
	(* Rückmeldung zu*)
	xRückIsClosed					:	BOOL;
	xInRükIsClosed					:	BOOL;
	xInRükIsClosedMb				:	BOOL;
	ITF_RükIsClosed					:	CtaSysIO.ITF_IO;
	(* Generelle Sicherung *)
    xFuseOk                     	:   BOOL;
    xInFuseOk                   	:   BOOL;
    xInFuseOkMb                 	:   BOOL;
	ITF_FuseOk 						:	CtaSysIO.ITF_IO;
 	(* Stellantriebs sicherung *)
    xActuatorFuseOk                	:   BOOL;    
    xInActuatorFuseOk              	:   BOOL;
    xInActuatorFuseOkMb            	:   BOOL;
	ITF_ActuatorFuseOk				:	CtaSysIO.ITF_IO;
	(* Ready signal *)
    xActuatorIsReady               	:   BOOL;
    xInActuatorIsReady             	:   BOOL;
    xInActuatorIsReadyMb           	:   BOOL;
	ITF_ActuatorIsReady				:	CtaSysIO.ITF_IO;
	(* Revisionsschalter *)
    xActuatorRevisionSwitchOn      	:   BOOL;
    xInActuatorRevisionSwitchOn    	:   BOOL;   
    xInActuatorRevisionSwitchOnMb   :   BOOL;
	ITF_RevisionSwitchOk			:	CtaSysIO.ITF_IO;	
	xActuatorRevisionSwitchOff		:	BOOL;
 	(* Hand Ansteuerung*)
    xActuatorHand                  	:   BOOL;
    xInActuatorHand                	:   BOOL;
    xInActuatorHandMb              	:   BOOL;
	ITF_ActuatorHand				:	CtaSysIO.ITF_IO; 
    (* Stellantrieb *)
    xReleaseFromModBus          	:   BOOL;
    xReleaseControllPrio        	:   BOOL;
    rReleaseFromModBus          	:   REAL;
    rReleaseControllPrio        	:   REAL;
    rReleaseScaled              	:   REAL;  
    xSafetyStopActuator       		:   BOOL := FALSE;  
  	(*Ventil Startöffnung*)
    TP_StartOeffnungVorlauf     	:   TP;
    (*Stellantrieb*)   
    fbStellantriebsMotor        	:   CtaSysMotor.fbMotor;  
    (* Modbus *)
    xModbusTest                 	:   BOOL;
    ayMbControllWord            	:   ARRAY[0..3] OF WORD;
    ayMbStateWord               	:   ARRAY[0..3] OF WORD;	
    (* Parameter *)	
    fbConfigFile					:   CtaSysConfig.fbConfigFile;
    scParameter                 	:   scParameter;	
    (* Reports *)	
    fbReportManager			    	:   CtaAppReport.fbReportManager;      
    difor					    	:	DINT;                                                                    
    ayErrorReporter					:	ARRAY[1..8] OF CtaAppReport.fbReporter;
	ayWarningReporter				:	ARRAY[1..4] OF CtaAppReport.fbReporter;    
	xErrorDiRük						:	BOOL;	(*Parametrierter Fehler DI*)	
	xErrorAIRük						:	BOOL;	(*Parametrierter Fehler AI*)
	xErrorDiffAI					:	BOOL;	(*Differenz von Stellwert zu Istwert*)
	xErrorOpenDI					:	BOOL;	(*Keine rückmeldung von Stellventil beim Öffnen*)
	xErrorCloseDI					:	BOOL;	(*Keine Rückmeldung von Stellventil beim Schlissen*)
	(* Trendlogs *)
	fbTrendxOnZu					:	CtaAppInfluxLog.FB_LOG_NODE_BOOL;
	fbTrendxRückClosed				:	CtaAppInfluxLog.FB_LOG_NODE_BOOL;
	fbTrendxOnAuf					:	CtaAppInfluxLog.FB_LOG_NODE_BOOL;
	fbTrendxRückIsOpen				:	CtaAppInfluxLog.FB_LOG_NODE_BOOL;
	fbTrendrOnY						:	CtaAppInfluxLog.FB_LOG_NODE_REAL;
	fbTrendrIsOnY					:	CtaAppInfluxLog.FB_LOG_NODE_REAL;
	fbTrendxError					:	CtaAppInfluxLog.FB_LOG_NODE_BOOL;
	(* Collector *)
    diArrayPosition					:   DINT;	
	(*Stellzeiten digitaler Stellantriebe*)
	rOnYOld							:	REAL;
	xEventOpen						:	BOOL;
	xEventClose						:	BOOL;
	tEventOpen						:	TIME;
	rAddEventOpen					:	REAL;
	rAddEventClose					:	REAL;
	tEventClose						:	TIME;
	TP_Open                			:   TP;
	TP_Close						:	TP; 
	(*Eingangsüberwachung Digital*)    	
	fbCheckRükOpen					:	CtaSysMotor.fbSafetyInput;
	fbCheckRükClosed				:	CtaSysMotor.fbSafetyInput;		
	(* Eingangsüberwachung Analog*)
	xStellwertOutOk					:	BOOL;
	xNoDiffAI						:	BOOL;
	fbCheckValueAI					:	CtaSysMotor.fbSafetyInput;		
	(*Überwachung Stellantrieb*)	
	xCheckRüAuf						:	BOOL;
	xCheclRüZu						:	BOOL;
END_VAR

(* Config *)
actConfig();

(* Motor Command *)
IF xIsEnabled AND NOT xConfigError THEN
    (* Modbus Controll *)
    actMbControll();
    (* Controll Prio *)
    actPrioOfControll();
	
	(*Startöffnung konfiguriert*)
	IF scParameter.scBase.fbxEnStartPosition.proValue THEN
		(*Verharrzeit konfiguriert*)
		IF scParameter.scBase.fbtStartPosTime.proValue > T#0MS THEN
			TP_StartOeffnungVorlauf(IN:= xReleaseControllPrio,PT := scParameter.scBase.fbtStartPosTime.proValue);
		END_IF	
	END_IF
	
	(*Übersteuerung mit YStartPos während Q von TP_StartOeffnungVorlauf*)
	rReleaseControllPrio := SEL(TP_StartOeffnungVorlauf.Q ,rReleaseControllPrio,scParameter.scBase.fbrYStartPos.proValue);
	
	(*Skalierung*)
    rReleaseScaled  :=  CtaAppBasic.fcScale(    rIn                 :=  rReleaseControllPrio,
                                                rMin                :=  0,
                                                rMax                :=  100,
                                                rOutMin             :=  scParameter.scBase.fbrYMin.proValue,
                                                rOutMax             :=  scParameter.scBase.fbrYMax.proValue);	
	(*Limitierung*)                                                        
    rReleaseScaled  := LIMIT(scParameter.scBase.fbrYMin.proValue , rReleaseScaled ,scParameter.scBase.fbrYMax.proValue);
    
    (* Motor *)                
    fbStellantriebsMotor     (   (* Inputs *)
                    xEn                 :=  xActuatorRevisionSwitchOn,
                    xFreigabe           :=  xReleaseControllPrio,
                    rFreigabeY          :=  rReleaseScaled,
                    xSafetyStop         :=  xSafetyStopActuator,
                    (* Parameter *)
                    fbxEnHandEin        :=  scParameter.scManual.fbxAlowManualOn,
                    fbxGeregelt         :=  scParameter.scBase.fbxRegulatet,
                    fbuiHandMode        :=  scParameter.scManual.fbuiManualState,
                    fbrStellwertHandY   :=  scParameter.scManual.fbrManualOnY,
                    (* Outputs *)
                    xOn                 =>  xOn,
                    rOnY                =>  ,
                    xHand               =>  );
	
	(* Dumping of the rOnY Value *)				
	fbDumperRonY(	xEn 	:=	xIsEnabled,
					rSoll	:=	SEL(xOn, scParameter.scBase.fbrYStopp.proValue, fbStellantriebsMotor.rOnY),
					rY		=>	rOnY);
                
	(*Invertierung*)
	IF scParameter.scBase.fbxInvertiert.proValue THEN
		rOnY := 100 - rOnY;
	END_IF
	
	(*Analogwert Überwachung*)
	IF scParameter.scInSAtActualPosition.fbxDoesAlarm.proValue > scParameter.scInSAtActualPosition.fbxEnable.proValue THEN		
		scParameter.scInSAtActualPosition.fbxDoesAlarm.proValue := FALSE;		
	END_IF
	
	IF scParameter.scInSAtActualPosition.fbxDoesAlarm.proValue THEN
		
		xStellwertOutOk := rOnY > 0;
	
		(*Überwachung der Stellwertabweichung*)
		IF rActualPosition > rOnY + scParameter.scInSAtActualPosition.fbrMaxDiff.proValue THEN
			xNoDiffAI	:=	FALSE;
		ELSIF rActualPosition < rOnY - scParameter.scInSAtActualPosition.fbrMaxDiff.proValue THEN
			xNoDiffAI	:=	FALSE;
		ELSIF rOnY = 0 THEN
			xNoDiffAI	:=	FALSE;
		ELSE
			xNoDiffAI :=	TRUE;
		END_IF

		fbCheckValueAI		(	(*Inputs*)
						xSafetyIn			:=	xNoDiffAI,	
						xReferenceIn		:=	xStellwertOutOk,	
						(*Parameter*)
						fbxEnSafetyInput	:=	scParameter.scInSAtActualPosition.fbxDoesAlarm,
						fbtStartTime		:=	scParameter.scInSAtActualPosition.fbtDelayStart,
						fbtRunTime			:=	scParameter.scInSAtActualPosition.fbtDelayRun,
						(*Fehler Output*)
						XError				=>	xErrorDiffAI);	
	END_IF
	
	IF scParameter.scBase.fbxEnDigitalValve.proValue THEN
		(*Stellzeiten bei Ventil mit Digitalen Ausängen*)
		IF scParameter.scBase.fbtYSettingTime.proValue > T#0S THEN
			IF rOnY > rOnYOld + scParameter.scBase.fbrHysteresisDigital.proValue THEN
				xEventOpen		:=	TRUE;
				xEventClose		:=	FALSE;
				(*Berrechnung der Öffnungszeit*)
				tEventOpen		:=	TO_TIME(TO_DINT((TO_REAL(TO_DINT(scParameter.scBase.fbtYSettingTime.proValue))/100) * (rOnY - rOnYOld + rAddEventOpen)));
				rAddEventOpen	:=	rAddEventOpen + rOnY - rOnYOld;
				rAddEventClose	:=	0.0;
				tEventClose		:=	T#0S;
				rOnYOld 		:=	rOnY;
			ELSIF rOnY < rOnYOld - scParameter.scBase.fbrHysteresisDigital.proValue THEN
				xEventClose		:=	TRUE;
				xEventOpen		:=	FALSE;
				(*Berrechnung der Schliesszeit*)
				tEventClose		:=	TO_TIME(TO_DINT((TO_REAL(TO_DINT(scParameter.scBase.fbtYSettingTime.proValue))/100) * (rOnYOld - rOnY + rAddEventClose)));
				rAddEventOpen	:=	0.0;
				rAddEventClose	:=	rAddEventClose + rOnYOld - rOnY;
				tEventOpen		:=	T#0S;
				rOnYOld			:=	rOnY;
			END_IF
			
			(*Ansteuerung Pulsgeber*)
			TP_Open		(IN		:=	xEventOpen AND NOT TP_Open.Q,
						 PT		:=	tEventOpen);
			TP_Close	(IN		:=	xEventClose AND NOT TP_Close.Q,
						 PT		:=	tEventClose);
						 
			(*Beschaltung der Ausgänge*)			 
			xOnAuf				:=	TP_Open.Q;
			xOnZu				:=	TP_Close.Q;
			
			IF TP_Close.Q OR TP_Open.Q THEN
				xEventOpen 		:=	FALSE;
				xEventClose		:=	FALSE;
			END_IF					 
		ELSE
			TP_Open.PT			:=	T#0S;
			TP_Close.PT			:=	T#0S;
			xOnAuf				:=	xOn;
			xOnZu				:=	NOT xOn;
		END_IF	
	END_IF
	
	(*Überwachung Eingangsrückmeldung*)
	
	IF scParameter.scInSAtRükOpen.fbxDoesAlarm.proValue > scParameter.scInSAtRükOpen.fbxEnable.proValue THEN
		scParameter.scInSAtRükOpen.fbxDoesAlarm.proValue := FALSE;		
	END_IF
		
	fbCheckRükOpen		(	(*Inputs*)
						xSafetyIn			:=	xRückIsOpen,	
						xReferenceIn		:=	xOnAuf,	
						(*Parameter*)
						fbxEnSafetyInput	:=	scParameter.scInSAtRükOpen.fbxDoesAlarm,
						fbtStartTime		:=	scParameter.scInSAtRükOpen.fbtDelayStart,
						fbtRunTime			:=	scParameter.scInSAtRükOpen.fbtDelayRun,
						(*Fehler Output*)
						XError				=>	xErrorOpenDI);
	(*Ventil- Rückmeldung offen*)
	IF scParameter.scInSAtRükOpen.fbxEnable.proValue THEN
		xIsOpen := xRückIsOpen; 
	ELSE
		xIsOpen := rOnY >= scParameter.scBase.fbrRefIsOpen.proValue;
	END_IF					
	
						
	IF scParameter.scInSAtRükClosed.fbxDoesAlarm.proValue > scParameter.scInSAtRükClosed.fbxEnable.proValue THEN
		scParameter.scInSAtRükClosed.fbxDoesAlarm.proValue := FALSE;		
	END_IF
	
	fbCheckRükClosed	(	(*Inputs*)
						xSafetyIn			:=	xRückIsClosed,	
						xReferenceIn		:=	xOnZu,	
						(*Parameter*)
						fbxEnSafetyInput	:=	scParameter.scInSAtRükClosed.fbxDoesAlarm,
						fbtStartTime		:=	scParameter.scInSAtRükClosed.fbtDelayStart,
						fbtRunTime			:=	scParameter.scInSAtRükClosed.fbtDelayRun,
						(*Fehler Output*)
						XError				=>	xErrorCloseDI);
						
	(*Ventil- Rückmeldung zu*)
	IF scParameter.scInSAtRükClosed.fbxEnable.proValue THEN
		xIsClose := xRückIsClosed;
	ELSE
		xIsClose := rOnY <= scParameter.scBase.fbrRefIsClosed.proValue;
	END_IF
							
	(*Monitoring nach eingestellten Parametern*)					
	xCheclRüZu			:=	FALSE;
	xCheckRüAuf			:=	FALSE;
	xErrorDiRük			:=	FALSE;
	xErrorAIRük			:=	FALSE;
	
	(*Monitoring*)
	IF scParameter.scBase.fbxEnDigitalMonitoring.proValue OR scParameter.scBase.fbxEnAnalogMonitoring.proValue THEN
		(*Prüfung des Stellwertes anhand eingestelleter Referenzen*)
		IF rOnY >= scParameter.scBase.fbrRefIsOpen.proValue THEN
			xCheckRüAuf	:=	TRUE;
		ELSIF rOnY <= scParameter.scBase.fbrRefIsClosed.proValue THEN
			xCheclRüZu	:=	TRUE;
		END_IF
		
		(*Monitoring der Digitalen Endopsition*)
		IF scParameter.scBase.fbxEnDigitalMonitoring.proValue THEN
			IF xCheckRüAuf THEN
				xErrorDiRük := NOT xRückIsOpen;
			ELSIF xCheclRüZu THEN
				xErrorDiRük := NOT xRückIsClosed;			
			END_IF
		END_IF
		
		(*Monitioring der Analogen Endposition*)			
		IF scParameter.scBase.fbxEnAnalogMonitoring.proValue THEN
			IF xCheckRüAuf THEN
				xErrorAIRük	:=	rActualPosition <= scParameter.scBase.fbrRefIsOpen.proValue;
			ELSIF xCheclRüZu THEN
				xErrorAIRük	:=	rActualPosition >= scParameter.scBase.fbrRefIsClosed.proValue;
			END_IF
		END_IF		
	END_IF   
	(* EWI *)
	actReport();
ELSE
    (* Off if Disabled or Config Error *)
    xOn  	:=	FALSE;
	xOnZu 	:=	FALSE;
	xOnAuf 	:=	FALSE;
    rOnY 	:=	0.0;
    
    (* Reset Flags *)
    actResetOnDisable();
	IF xConfigError THEN
		(*EWI*)
		actReport();
	END_IF
END_IF;

(* State *)
actState();
(* Modbus State *)
actMbState();
(* InfluxDB *)
actTrendLog();

PROPERTY proHandOn : BOOL
SET
IF proHandOn THEN
    scParameter.scManual.fbuiManualState.proValue := 2;
END_IF;
END_SET
GET
proHandOn := xIsHandOn;
END_GET
END_PROPERTY

PROPERTY proAuto : BOOL
SET
IF proAuto THEN
    scParameter.scManual.fbuiManualState.proValue := 0;
END_IF;
END_SET
GET
proAuto := xIsAuto;
END_GET
END_PROPERTY

PROPERTY proHandOff : BOOL
SET
IF proHandOff THEN
    scParameter.scManual.fbuiManualState.proValue := 1;
END_IF;
END_SET
GET
proHandOff := xIsHandOff;
END_GET
END_PROPERTY

PROPERTY proHandOnY : REAL
SET
scParameter.scManual.fbrManualOnY.proValue := proHandOnY;
END_SET
GET
proHandOnY := scParameter.scManual.fbrManualOnY.proValue;
END_GET
END_PROPERTY

PROPERTY proHardWareHandModulAktive : BOOL
GET
proHardWareHandModulAktive := xActuatorHand;
END_GET
END_PROPERTY

ACTION actConfig:
(* Config Fb *)
fbConfigFile();

(* Base Parameter *)
scParameter.scBase.fbxEnable                				(_usiParaNr :=  1, ItfConfigFb := fbConfigFile);
scParameter.scBase.fbxRegulatet             				(_usiParaNr :=  2, ItfConfigFb := fbConfigFile);
scParameter.scBase.fbxControllMb            				(_usiParaNr :=  3, ItfConfigFb := fbConfigFile);
scParameter.scBase.fbxInvertiert							(_usiParaNr :=	4, itfConfigFb := fbConfigFile);
scParameter.scBase.fbrYMin                  				(_usiParaNr :=  5, ItfConfigFb := fbConfigFile);
scParameter.scBase.fbrYMax                  				(_usiParaNr :=  6, ItfConfigFb := fbConfigFile);
scParameter.scBase.fbxEnStartPosition						(_usiParaNr :=  7, ItfConfigFb := fbConfigFile);
scParameter.scBase.fbrYStartPos								(_usiParaNr :=  8, itfConfigFb := fbConfigFile);
scParameter.scBase.fbtStartPosTime							(_usiParaNr :=  9, itfConfigFb := fbConfigFile);
scParameter.scBase.fbrYStopp								(_usiParaNr := 10, itfConfigFb := fbConfigFile);
scParameter.scBase.fbtYSettingTime							(_usiParaNr := 11, itfConfigFb := fbConfigFile);
scParameter.scBase.fbxEnDigitalValve						(_usiParaNr := 12, itfConfigFb := fbConfigFile);
scParameter.scBase.fbrHysteresisDigital						(_usiParaNr := 13, itfConfigFb := fbConfigFile);
scParameter.scBase.fbrRefIsOpen								(_usiParaNr := 14, itfConfigFb := fbConfigFile);
scParameter.scBase.fbrRefIsClosed							(_usiParaNr := 15, itfConfigFb := fbConfigFile);
scParameter.scBase.fbxEnDigitalMonitoring					(_usiParaNr := 16, itfConfigFb := fbConfigFile);
scParameter.scBase.fbxEnAnalogMonitoring					(_usiParaNr := 17, itfConfigFb := fbConfigFile);
                                                        	
(* Fuse Parameter *)                                    	
scParameter.scFuse.fbxEnable                				(_usiParaNr := 18, ItfConfigFb := fbconfigFile);
scParameter.scFuse.fbxInputMb               				(_usiParaNr := 19, ItfConfigFb := fbconfigFile);
scParameter.scFuse.fbxDoesAlarm             				(_usiParaNr := 20, ItfConfigFb := fbconfigFile);
                                                        	
(* Stellantrieb Fuse Parameter *)                       	
scParameter.scActuatorFuse.fbxEnable           				(_usiParaNr := 21, ItfConfigFb := fbconfigFile);
scParameter.scActuatorFuse.fbxInputMb          				(_usiParaNr := 22, ItfConfigFb := fbconfigFile);
scParameter.scActuatorFuse.fbxDoesAlarm        				(_usiParaNr := 23, ItfConfigFb := fbconfigFile);
                                                        	
(* Revision Switch Parameter *)                         	
scParameter.scInSAtRevisionSwitch.fbxEnable  				(_usiParaNr := 24, ItfConfigFb := fbconfigFile);
scParameter.scInSAtRevisionSwitch.fbxInputMb 				(_usiParaNr := 25, ItfConfigFb := fbconfigFile);
                                                        	
(* Ready Input Parameter *)                             	
scParameter.scInSAtReady.fbxEnable           				(_usiParaNr := 26, ItfConfigFb := fbconfigFile);
scParameter.scInSAtReady.fbxInputMb          				(_usiParaNr := 27, ItfConfigFb := fbconfigFile);
                                                        	
(* Stellantrieb Input Hand *)                           	
scParameter.scInSAtHand.fbxEnable            				(_usiParaNr := 28, ItfConfigFb := fbconfigFile);
scParameter.scInSAtHand.fbxInputMb           				(_usiParaNr := 29, ItfConfigFb := fbconfigFile);
                                                        	
(* Is closed Input Parameter *)                         	
scParameter.scInSAtRükClosed.fbxEnable		 				(_usiParaNr := 30, ItfConfigFb := fbconfigFile);             
scParameter.scInSAtRükClosed.fbxInputMb      				(_usiParaNr := 31, ItfConfigFb := fbconfigFile);
scParameter.scInSAtRükClosed.fbxDoesAlarm    				(_usiParaNr := 32, ItfConfigFb := fbconfigFile);
scParameter.scInSAtRükClosed.fbtDelayStart   				(_usiParaNr := 33, ItfConfigFb := fbconfigFile);
scParameter.scInSAtRükClosed.fbtDelayRun     				(_usiParaNr := 34, ItfConfigFb := fbconfigFile);
scParameter.scInSAtRükClosed.fbiTypeOfAck					(_usiParaNr := 35, itfConfigFb := fbConfigFile,_MinInit := 0,_MaxInit :=2);
scParameter.scInSAtRükClosed.fbiMaxErrorRetryAllowed		(_usiParaNr := 36 , itfConfigFb := fbConfigFile);
                                                        	
(* Is open Input Parameter *)                           	
scParameter.scInSAtRükOpen.fbxEnable		 				(_usiParaNr := 37, ItfConfigFb := fbconfigFile);             
scParameter.scInSAtRükOpen.fbxInputMb        				(_usiParaNr := 38, ItfConfigFb := fbconfigFile);
scParameter.scInSAtRükOpen.fbxDoesAlarm      				(_usiParaNr := 39, ItfConfigFb := fbconfigFile);
scParameter.scInSAtRükOpen.fbtDelayStart     				(_usiParaNr := 40, ItfConfigFb := fbconfigFile);
scParameter.scInSAtRükOpen.fbtDelayRun       				(_usiParaNr := 41, ItfConfigFb := fbconfigFile);
scParameter.scInSAtRükOpen.fbiTypeOfAck						(_usiParaNr := 42, itfConfigFb := fbConfigFile,_MinInit := 0,_MaxInit :=2);
scParameter.scInSAtRükOpen.fbiMaxErrorRetryAllowed			(_usiParaNr := 43, itfConfigFb := fbConfigFile);
                                                        	
(* Actual value Input Parameter *)                      	
scParameter.scInSAtActualPosition.fbxEnable     			(_usiParaNr := 44, ItfConfigFb := fbconfigFile);
scParameter.scInSAtActualPosition.fbxInputMb    			(_usiParaNr := 45, ItfConfigFb := fbconfigFile);
scParameter.scInSAtActualPosition.fbxDoesAlarm  			(_usiParaNr := 46, ItfConfigFb := fbconfigFile);
scParameter.scInSAtActualPosition.fbrMaxDiff    			(_usiParaNr := 47, ItfConfigFb := fbconfigFile);
scParameter.scInSAtActualPosition.fbtDelayStart 			(_usiParaNr := 48, ItfConfigFb := fbconfigFile);
scParameter.scInSAtActualPosition.fbtDelayRun   			(_usiParaNr := 49, ItfConfigFb := fbconfigFile);
scParameter.scInSAtActualPosition.fbiTypeOfAck				(_usiParaNr := 50, itfConfigFb := fbConfigFile,_MinInit := 0,_MaxInit :=2);
scParameter.scInSAtActualPosition.fbiMaxErrorRetryAllowed	(_usiParaNr := 51, itfConfigFb := fbConfigFile);

(* InfluxDb *)
scParameter.scInfluxDb.fbxEnable            				(_usiParaNr := 52, ItfConfigFb := fbconfigFile);
                                                        	
(* Manual Parameter *)                                  	
scParameter.scManual.fbxAlowManualOn        				(_usiParaNr := 53, ItfConfigFb := fbconfigFile); 
scParameter.scManual.fbuiManualState        				(_usiParaNr := 54, ItfConfigFb := fbconfigFile);
scParameter.scManual.fbrManualOnY           				(_usiParaNr := 55, ItfConfigFb := fbconfigFile);

xConfigError := fbConfigFile.xError;
END_ACTION

PROPERTY p_scInfluxDb_fbxEnable : CtaSysConfig.ITF_DATATYPE;
GET
p_scInfluxDb_fbxEnable := scParameter.scInfluxDb.fbxEnable;
END_GET
END_PROPERTY

PROPERTY p_scActuatorFuse_fbxEnable : CtaSysConfig.ITF_DATATYPE;
GET
p_scActuatorFuse_fbxEnable := scParameter.scActuatorFuse.fbxEnable;
END_GET
END_PROPERTY

PROPERTY p_scActuatorFuse_fbxInputMb : CtaSysConfig.ITF_DATATYPE;
GET
p_scActuatorFuse_fbxInputMb := scParameter.scActuatorFuse.fbxInputMb;
END_GET
END_PROPERTY

PROPERTY p_scActuatorFuse_fbxDoesAlarm : CtaSysConfig.ITF_DATATYPE;
GET
p_scActuatorFuse_fbxDoesAlarm := scParameter.scActuatorFuse.fbxDoesAlarm;
END_GET
END_PROPERTY

PROPERTY p_scBase_fbxEnable : CtaSysConfig.ITF_DATATYPE;
GET
p_scBase_fbxEnable := scParameter.scBase.fbxEnable;
END_GET
END_PROPERTY

PROPERTY p_scBase_fbxControllMb : CtaSysConfig.ITF_DATATYPE;
GET
p_scBase_fbxControllMb := scParameter.scBase.fbxControllMb ;
END_GET
END_PROPERTY

PROPERTY p_scBase_fbxInvertiert : CtaSysConfig.ITF_DATATYPE;
GET
p_scBase_fbxInvertiert := scParameter.scBase.fbxInvertiert;
END_GET
END_PROPERTY

PROPERTY p_scBase_fbxRegulatet : CtaSysConfig.ITF_DATATYPE;
GET
p_scBase_fbxRegulatet := scParameter.scBase.fbxRegulatet;
END_GET
END_PROPERTY

PROPERTY p_scBase_fbrYMin : CtaSysConfig.ITF_DATATYPE;
GET
p_scBase_fbrYMin := scParameter.scBase.fbrYMin;
END_GET
END_PROPERTY

PROPERTY p_scBase_fbrYMax : CtaSysConfig.ITF_DATATYPE;
GET
p_scBase_fbrYMax := scParameter.scBase.fbrYMax;
END_GET
END_PROPERTY

PROPERTY p_scBase_fbxEnStartPosition : CtaSysConfig.ITF_DATATYPE;
GET
p_scBase_fbxEnStartPosition := scParameter.scBase.fbxEnStartPosition;
END_GET
END_PROPERTY

PROPERTY p_scBase_fbrYStartPos : CtaSysConfig.ITF_DATATYPE;
GET
p_scBase_fbrYStartPos := scParameter.scBase.fbrYStartPos;
END_GET
END_PROPERTY

PROPERTY p_scBase_fbtStartPosTime : CtaSysConfig.ITF_DATATYPE;
GET
p_scBase_fbtStartPosTime := scParameter.scBase.fbtStartPosTime;
END_GET
END_PROPERTY

PROPERTY p_scBase_fbrYStopp : CtaSysConfig.ITF_DATATYPE;
GET
p_scBase_fbrYStopp := scParameter.scBase.fbrYStopp;
END_GET
END_PROPERTY

PROPERTY p_scBase_fbtYSettingTime : CtaSysConfig.ITF_DATATYPE;
GET
p_scBase_fbtYSettingTime := scParameter.scBase.fbtYSettingTime;
END_GET
END_PROPERTY

PROPERTY p_scBase_fbxEnDigitalValve : CtaSysConfig.ITF_DATATYPE;
GET
p_scBase_fbxEnDigitalValve := scParameter.scBase.fbxEnDigitalValve;
END_GET
END_PROPERTY

PROPERTY p_scBase_fbrHysteresisDigital : CtaSysConfig.ITF_DATATYPE;
GET
p_scBase_fbrHysteresisDigital := scParameter.scBase.fbrHysteresisDigital;
END_GET
END_PROPERTY

PROPERTY p_scBase_fbrRefIsOpen : CtaSysConfig.ITF_DATATYPE;
GET
p_scBase_fbrRefIsOpen := scParameter.scBase.fbrRefIsOpen;
END_GET
END_PROPERTY

PROPERTY p_scBase_fbrRefIsClosed : CtaSysConfig.ITF_DATATYPE;
GET
p_scBase_fbrRefIsClosed := scParameter.scBase.fbrRefIsClosed;
END_GET
END_PROPERTY

PROPERTY p_scBase_fbxEnDigitalMonitoring : CtaSysConfig.ITF_DATATYPE;
GET
p_scBase_fbxEnDigitalMonitoring := scParameter.scBase.fbxEnDigitalMonitoring;
END_GET
END_PROPERTY

PROPERTY p_scBase_fbxEnAnalogMonitoring : CtaSysConfig.ITF_DATATYPE;
GET
p_scBase_fbxEnAnalogMonitoring := scParameter.scBase.fbxEnAnalogMonitoring;
END_GET
END_PROPERTY

PROPERTY p_scFuse_fbxEnable : CtaSysConfig.ITF_DATATYPE;
GET
p_scFuse_fbxEnable := scParameter.scFuse.fbxEnable;
END_GET
END_PROPERTY

PROPERTY p_scFuse_fbxInputMb : CtaSysConfig.ITF_DATATYPE;
GET
p_scFuse_fbxInputMb := scParameter.scFuse.fbxInputMb;
END_GET
END_PROPERTY

PROPERTY p_scFuse_fbxDoesAlarm : CtaSysConfig.ITF_DATATYPE;
GET
p_scFuse_fbxDoesAlarm := scParameter.scFuse.fbxDoesAlarm ;
END_GET
END_PROPERTY

PROPERTY p_scInStellAtRevisionSwitch_fbxEnable : CtaSysConfig.ITF_DATATYPE;
GET
p_scInStellAtRevisionSwitch_fbxEnable := scParameter.scInSAtRevisionSwitch.fbxEnable;
END_GET
END_PROPERTY

PROPERTY p_scInStellAtRevisionSwitch_fbxInputMb : CtaSysConfig.ITF_DATATYPE;
GET
p_scInStellAtRevisionSwitch_fbxInputMb := scParameter.scInSAtRevisionSwitch.fbxInputMb;
END_GET
END_PROPERTY

PROPERTY p_scInStellAtReady_fbxEnable : CtaSysConfig.ITF_DATATYPE;
GET
p_scInStellAtReady_fbxEnable := scParameter.scInSAtReady.fbxEnable;
END_GET
END_PROPERTY

PROPERTY p_scInStellAtReady_fbxInputMb : CtaSysConfig.ITF_DATATYPE;
GET
p_scInStellAtReady_fbxInputMb := scParameter.scInSAtReady.fbxInputMb;
END_GET
END_PROPERTY

PROPERTY p_scInStellAtHand_fbxEnable : CtaSysConfig.ITF_DATATYPE;
GET
p_scInStellAtHand_fbxEnable := scParameter.scInSAtHand.fbxEnable;
END_GET
END_PROPERTY

PROPERTY p_scInStellAtHand_fbxInputMb : CtaSysConfig.ITF_DATATYPE;
GET
p_scInStellAtHand_fbxInputMb := scParameter.scInSAtHand.fbxInputMb;
END_GET
END_PROPERTY

PROPERTY p_scInStellAtRükClosed_fbxEnable : CtaSysConfig.ITF_DATATYPE;
GET
p_scInStellAtRükClosed_fbxEnable := scParameter.scInSAtRükClosed.fbxEnable;
END_GET
END_PROPERTY

PROPERTY p_scInStellAtRükClosed_fbxInputMb : CtaSysConfig.ITF_DATATYPE;
GET
p_scInStellAtRükClosed_fbxInputMb := scParameter.scInSAtRükClosed.fbxInputMb;
END_GET
END_PROPERTY

PROPERTY p_scInStellAtRükClosed_fbxDoesAlarm : CtaSysConfig.ITF_DATATYPE;
GET
p_scInStellAtRükClosed_fbxDoesAlarm := scParameter.scInSAtRükClosed.fbxDoesAlarm;
END_GET
END_PROPERTY

PROPERTY p_scInStellAtRükClosed_fbtDelayStart : CtaSysConfig.ITF_DATATYPE;
GET
p_scInStellAtRükClosed_fbtDelayStart := scParameter.scInSAtRükClosed.fbtDelayStart;
END_GET
END_PROPERTY

PROPERTY p_scInStellAtRükClosed_fbtDelayRun : CtaSysConfig.ITF_DATATYPE;
GET
p_scInStellAtRükClosed_fbtDelayRun := scParameter.scInSAtRükClosed.fbtDelayRun;
END_GET
END_PROPERTY

PROPERTY p_scInStellAtRükClosed_fbiTypeOfAck : CtaSysConfig.ITF_DATATYPE;
GET
p_scInStellAtRükClosed_fbiTypeOfAck := scParameter.scInSAtRükClosed.fbiTypeOfAck;
END_GET
END_PROPERTY

PROPERTY p_scInStellAtRükClosed_fbiMaxErrorRetryAllowed : CtaSysConfig.ITF_DATATYPE;
GET
p_scInStellAtRükClosed_fbiMaxErrorRetryAllowed := scParameter.scInSAtRükClosed.fbiMaxErrorRetryAllowed;
END_GET
END_PROPERTY

PROPERTY p_scInStellAtRükOpen_fbxEnable : CtaSysConfig.ITF_DATATYPE;
GET
p_scInStellAtRükOpen_fbxEnable := scParameter.scInSAtRükOpen.fbxEnable;
END_GET
END_PROPERTY

PROPERTY p_scInStellAtRükOpen_fbxInputMb : CtaSysConfig.ITF_DATATYPE;
GET
p_scInStellAtRükOpen_fbxInputMb := scParameter.scInSAtRükOpen.fbxInputMb;
END_GET
END_PROPERTY

PROPERTY p_scInStellAtRükOpen_fbxDoesAlarm : CtaSysConfig.ITF_DATATYPE;
GET
p_scInStellAtRükOpen_fbxDoesAlarm := scParameter.scInSAtRükOpen.fbxDoesAlarm;
END_GET
END_PROPERTY

PROPERTY p_scInStellAtRükOpen_fbtDelayStart : CtaSysConfig.ITF_DATATYPE;
GET
p_scInStellAtRükOpen_fbtDelayStart := scParameter.scInSAtRükOpen.fbtDelayStart;
END_GET
END_PROPERTY

PROPERTY p_scInStellAtRükOpen_fbtDelayRun : CtaSysConfig.ITF_DATATYPE;
GET
p_scInStellAtRükOpen_fbtDelayRun := scParameter.scInSAtRükOpen.fbtDelayRun;
END_GET
END_PROPERTY

PROPERTY p_scInStellAtRükOpen_fbiTypeOfAck : CtaSysConfig.ITF_DATATYPE;
GET
p_scInStellAtRükOpen_fbiTypeOfAck := scParameter.scInSAtRükOpen.fbiTypeOfAck;
END_GET
END_PROPERTY

PROPERTY p_scInStellAtRükOpen_fbiMaxErrorRetryAllowed : CtaSysConfig.ITF_DATATYPE;
GET
p_scInStellAtRükOpen_fbiMaxErrorRetryAllowed := scParameter.scInSAtRükOpen.fbiMaxErrorRetryAllowed;
END_GET
END_PROPERTY

PROPERTY p_scInStellAtActualPosition_fbxEnable : CtaSysConfig.ITF_DATATYPE;
GET
p_scInStellAtActualPosition_fbxEnable := scParameter.scInSAtActualPosition.fbxEnable;
END_GET
END_PROPERTY

PROPERTY p_scInStellAtActualPosition_fbxInputMb : CtaSysConfig.ITF_DATATYPE;
GET
p_scInStellAtActualPosition_fbxInputMb := scParameter.scInSAtActualPosition.fbxInputMb;
END_GET
END_PROPERTY

PROPERTY p_scInStellAtActualPosition_fbxDoesAlarm : CtaSysConfig.ITF_DATATYPE;
GET
p_scInStellAtActualPosition_fbxDoesAlarm := scParameter.scInSAtActualPosition.fbxDoesAlarm;
END_GET
END_PROPERTY

PROPERTY p_scInStellAtActualPosition_fbrMaxDiff : CtaSysConfig.ITF_DATATYPE;
GET
p_scInStellAtActualPosition_fbrMaxDiff := scParameter.scInSAtActualPosition.fbrMaxDiff;
END_GET
END_PROPERTY

PROPERTY p_scInStellAtActualPosition_fbtDelayStart : CtaSysConfig.ITF_DATATYPE;
GET
p_scInStellAtActualPosition_fbtDelayStart := scParameter.scInSAtActualPosition.fbtDelayStart;
END_GET
END_PROPERTY

PROPERTY p_scInStellAtActualPosition_fbtDelayRun : CtaSysConfig.ITF_DATATYPE;
GET
p_scInStellAtActualPosition_fbtDelayRun := scParameter.scInSAtActualPosition.fbtDelayRun;
END_GET
END_PROPERTY

PROPERTY p_scInStellAtActualPosition_fbiTypeOfAck : CtaSysConfig.ITF_DATATYPE;
GET
p_scInStellAtActualPosition_fbiTypeOfAck := scParameter.scInSAtActualPosition.fbiTypeOfAck;
END_GET
END_PROPERTY

PROPERTY p_scInStellAtActualPosition_fbiMaxErrorRetryAllowed : CtaSysConfig.ITF_DATATYPE;
GET
p_scInStellAtActualPosition_fbiMaxErrorRetryAllowed := scParameter.scInSAtActualPosition.fbiMaxErrorRetryAllowed;
END_GET
END_PROPERTY

PROPERTY p_scManual_fbxAlowManualOn : CtaSysConfig.ITF_DATATYPE;
GET
p_scManual_fbxAlowManualOn := scParameter.scManual.fbxAlowManualOn;
END_GET
END_PROPERTY

PROPERTY p_scManual_fbuiManualState : CtaSysConfig.ITF_DATATYPE;
GET
p_scManual_fbuiManualState := scParameter.scManual.fbuiManualState;
END_GET
END_PROPERTY

PROPERTY p_scManual_fbrManualOnY : CtaSysConfig.ITF_DATATYPE;
GET
p_scManual_fbrManualOnY := scParameter.scManual.fbrManualOnY;
END_GET
END_PROPERTY

PROPERTY proRefToRonYDumper : REFERENCE TO CtaAppDumper.fbDumper
GET
proRefToRonYDumper REF= fbDumperRonY;
END_GET
END_PROPERTY

PROPERTY proConfigError : BOOL
GET
proConfigError := xConfigError;
END_GET
END_PROPERTY

PROPERTY proValveIcon : UINT
GET
proValveIcon := uiValveIcon;
END_GET
SET
uiValveIcon := proValveIcon;
END_SET
END_PROPERTY

ACTION actMbControll:
IF NOT xModbusTest THEN
    (* Controll Word 0 Digital Controll *)
    (* Release from Modbus *)
    IF scParameter.scBase.fbxControllMb.proValue THEN
        xReleaseFromModBus              := ayMbControllWord[0].0; 
        (* Controll Word 1 setpoint*)
        rReleaseFromModBus              := LIMIT(0,TO_REAL(TO_INT(ayMbControllWord[1]))/10,100);   
    ELSE
        xReleaseFromModBus              := FALSE;
        rReleaseFromModBus              := 0; 
    END_IF;
    (* Actuator Ready *)
    IF scParameter.scInSAtReady.fbxInputMb.proValue THEN
        xInActuatorIsReadyMb               := ayMbControllWord[0].2;
    ELSE
        xInActuatorIsReadyMb               := FALSE;
    END_IF;
    (* Actuator is Open *)
   	IF scParameter.scInSAtRükOpen.fbxInputMb.proValue THEN
        xInRükIsOpenMb                  := ayMbControllWord[0].3;
    ELSE
        xInRükIsOpenMb                  := FALSE;
    END_IF; 
    (* Actuator is Closed *)
    IF scParameter.scInSAtRükClosed.fbxInputMb.proValue THEN
        xInRükIsClosedMb               := ayMbControllWord[0].4;
    ELSE
        xInRükIsClosedMb               := FALSE;
    END_IF;
    (* Revision Switch *)
    IF scParameter.scInSAtRevisionSwitch.fbxInputMb.proValue THEN
        xInActuatorRevisionSwitchOnMb      := ayMbControllWord[0].5;
    ELSE
        xInActuatorRevisionSwitchOnMb      := FALSE;    
    END_IF;
    (* Fuse Ok *)
    IF scParameter.scFuse.fbxInputMb.proValue THEN    
        xInFuseOkMb                     := ayMbControllWord[0].6;
    ELSE
        xInFuseOkMb                     := FALSE;
    END_IF;
    (* Actuator Protection *)
    IF scParameter.scActuatorFuse.fbxInputMb.proValue THEN
        xInActuatorFuseOkMb                := ayMbControllWord[0].7;
    ELSE
        xInActuatorFuseOkMb                := FALSE;
    END_IF;
    (* Actuator Hand *)
    IF scParameter.scInSAtHand.fbxInputMb.proValue THEN
        xInActuatorHandMb                  := ayMbControllWord[0].8;
    ELSE
        xInActuatorHandMb                  := FALSE;
    END_IF; 
	(* Actual Position*)
	IF scParameter.scInSAtActualPosition.fbxInputMb.proValue THEN
		rInActualPositionMb					:= LIMIT(0,TO_REAL(TO_INT(ayMbControllWord[2]))/10,100);
	ELSE  
		rInActualPositionMb					:= 0; 
	END_IF
ELSE
    xReleaseFromModBus              	:= FALSE;
    rReleaseFromModBus              	:= 0;     
    xInActuatorIsReadyMb               	:= FALSE;
	xInRükIsOpenMb						:= FALSE;
	xInRükIsClosedMb					:= FALSE;
    xInActuatorRevisionSwitchOnMb      	:= FALSE; 
    xInFuseOkMb                     	:= FALSE;
    xInActuatorFuseOkMb                	:= FALSE;
    xInActuatorHandMb                  	:= FALSE;
	rInActualPositionMb					:= 0;
END_IF;
END_ACTION

ACTION actMbState:
IF NOT xModbusTest THEN
    (* State Word 0 Digital Info*)
    ayMbStateWord[0].00     := xOnAuf;
    ayMbStateWord[0].01     := xOnZu;
    ayMbStateWord[0].02     := xActuatorIsReady;
    ayMbStateWord[0].03     := xRückIsOpen;
    ayMbStateWord[0].04     := xRückIsClosed;
    ayMbStateWord[0].05     := xActuatorRevisionSwitchOn;
    ayMbStateWord[0].06     := xFuseOk;
    ayMbStateWord[0].07     := xActuatorFuseOk;
    ayMbStateWord[0].08     := xIsHand;
    ayMbStateWord[0].09     := xIsAuto;
    ayMbStateWord[0].10     := FALSE;
    ayMbStateWord[0].11     := FALSE;
    ayMbStateWord[0].12     := FALSE;
    ayMbStateWord[0].13     := FALSE;
    ayMbStateWord[0].14     := xIsWarning;
    ayMbStateWord[0].15     := xIsError;
    (* State Word 1 setpoint*)
    ayMbStateWord[1]        := TO_WORD((TO_INT(rOnY * 10)));
    (* State Word 2 actual value*)
    ayMbStateWord[2]        := SEL(scParameter.scInSAtActualPosition.fbxEnable.proValue,TO_WORD((TO_INT(rOnY * 10))),TO_WORD((TO_INT(rActualPosition * 10))));
END_IF;
END_ACTION

PROPERTY proModbusTest : BOOL
SET
xModbusTest := proModbusTest;
END_SET
GET
proModbusTest := xModbusTest;
END_GET
END_PROPERTY

PROPERTY proModbusStateWord : REFERENCE TO ARRAY[0..3] OF WORD
GET
proModbusStateWord REF= ayMbStateWord;
END_GET
END_PROPERTY

PROPERTY proModbusControllWord : REFERENCE TO ARRAY[0..3] OF WORD
GET
proModbusControllWord REF= ayMbControllWord;
END_GET
END_PROPERTY

PROPERTY proIsError : BOOL
GET
proIsError := xIsError;
END_GET
END_PROPERTY

PROPERTY proIsWarning : BOOL
GET
proIsWarning := xIsWarning;
END_GET
END_PROPERTY

PROPERTY proIsRegulatet : BOOL
GET
proIsRegulatet := xIsRegulatet;
END_GET
END_PROPERTY

PROPERTY proIsEnabled : BOOL
GET
proIsEnabled := xIsEnabled;
END_GET
END_PROPERTY

ACTION actState:
xIsWarning        := _xIsWarning;         
xIsError          := _xIsError;          
xIsRegulatet      := scParameter.scBase.fbxRegulatet.proValue;         
xIsEnabled        := scParameter.scBase.fbxEnable.proValue;
xIsInverted		  := scParameter.scBase.fbxInvertiert.proValue; 
xIsHandOn         := scParameter.scManual.fbuiManualState.proValue = 2;         
xIsHandOff        := scParameter.scManual.fbuiManualState.proValue = 1;          
xIsAuto           := scParameter.scManual.fbuiManualState.proValue = 0 AND NOT xActuatorHand;  
xIsHand           := xIsHandOn OR xIsHandOff OR xActuatorHand;
END_ACTION

PROPERTY proIsHandOnOrOff : BOOL
GET
proIsHandOnOrOff := xIsHand;
END_GET
END_PROPERTY

PROPERTY proIsReady : BOOL
GET
proIsReady := xActuatorIsReady AND NOT xIsError;
END_GET
END_PROPERTY

PROPERTY proIsOnY : REAL
GET
proIsOnY := rActualPosition;
END_GET
END_PROPERTY

PROPERTY proRevisionSwitchOk : BOOL
GET
proRevisionSwitchOk := xActuatorRevisionSwitchOn;
END_GET
END_PROPERTY

PROPERTY proStateSymbol : STRING
GET
IF xIsError THEN
    proStateSymbol := 'CtaVisSymbols.ImagePool.CtaError';
ELSE    
    IF xIsWarning THEN
        IF scEWI.iWarning = 2 THEN
            proStateSymbol := 'CtaVisSymbols.ImagePool.front_hand_Yellow_Off';
        ELSIF scEWI.iWarning = 3 THEN
            proStateSymbol := 'CtaVisSymbols.ImagePool.front_hand_Yellow';
        ELSE
            proStateSymbol := 'CtaVisSymbols.ImagePool.CtaWarning';
        END_IF;
     ELSE
         proStateSymbol := '';
	 END_IF
END_IF;
END_GET
END_PROPERTY

PROPERTY proAnzError : INT
GET
proAnzError := fbReportManager.proAnzError;
END_GET
END_PROPERTY

PROPERTY proAnzInfo : INT
GET
proAnzInfo := fbReportManager.proAnzInfo;
END_GET
END_PROPERTY

PROPERTY proAnzWarning : INT
GET
proAnzWarning := fbReportManager.proAnzWarning;
END_GET
END_PROPERTY

PROPERTY proITF_REPORTMANAGER : CtaAppReport.ITF_REPORTMANAGER
GET
proITF_REPORTMANAGER := fbReportManager;
END_GET
END_PROPERTY

PROPERTY proIsInverted : BOOL
GET
proIsInverted := xIsInverted;
END_GET
END_PROPERTY

PROPERTY proRükIsClosed : BOOL
GET
proRükIsClosed := xRückIsClosed;
END_GET
END_PROPERTY

PROPERTY proRükIsOpen : BOOL
GET
proRükIsOpen := xRückIsOpen;
END_GET
END_PROPERTY

PROPERTY proOn : BOOL
GET
proOn := xReleaseControllPrio;
END_GET
END_PROPERTY

METHOD metDI_RükIsOpen
VAR_INPUT
    ITF_IN		:	CtaSysIO.ITF_IO;
END_VAR
VAR	
	ITF_DI		:	CtaSysIO.ITF_DI;
END_VAR
IF ITF_IN <> 0 THEN
	ITF_RükIsOpen := ITF_IN;
	IF __QUERYINTERFACE(ITF_RükIsOpen,ITF_DI) THEN
		xInRükIsOpen := ITF_DI.proValue;
	END_IF
ELSE
	xInRükIsOpen := 0;
END_IF
END_METHOD

PROPERTY proGetDI_RükIsOpen : BOOL
GET
proGetDI_RükIsOpen := xInRükIsOpen;
END_GET
END_PROPERTY

PROPERTY proNotShowDI_RükIsOpen : BOOL
GET
proNotShowDI_RükIsOpen := NOT scParameter.scInSAtRükOpen.fbxEnable.xValue OR scParameter.scInSAtRükOpen.fbxInputMb.xValue;
END_GET
END_PROPERTY

PROPERTY proIsOpen_ITF : CtaSysIO.ITF_IO
GET
proIsOpen_ITF := ITF_RükIsOpen;
END_GET
END_PROPERTY

METHOD metDI_RükIsClosed
VAR_INPUT
    ITF_IN		:	CtaSysIO.ITF_IO;
END_VAR
VAR	
	ITF_DI		:	CtaSysIO.ITF_DI;
END_VAR
IF ITF_IN <> 0 THEN
	ITF_RükIsClosed := ITF_IN;
	IF __QUERYINTERFACE(ITF_RükIsClosed,ITF_DI) THEN
		xInRükIsClosed := ITF_DI.proValue;
	END_IF
ELSE
	xInRükIsClosed := 0;
END_IF
END_METHOD

PROPERTY proGetDI_RükIsClosed : BOOL
GET
proGetDI_RükIsClosed := xInRükIsClosed;
END_GET
END_PROPERTY

PROPERTY proNotShowDI_RükIsClosed : BOOL
GET
proNotShowDI_RükIsClosed := NOT scParameter.scInSAtRükClosed.fbxEnable.xValue OR scParameter.scInSAtRükClosed.fbxInputMb.xValue;
END_GET
END_PROPERTY

PROPERTY proIsClosed_ITF : CtaSysIO.ITF_IO
GET
proIsClosed_ITF := ITF_RükIsClosed;
END_GET
END_PROPERTY

